LIN {X 0,Y 531.689,Z 306.036,A -85,B 0,C 180,E1 -12408.025,E2 -12408.025} C_VEL
LIN {X 0,Y 532.724,Z 312.75,A -85,B 0,C 180,E1 -12409.009,E2 -12409.009} C_VEL
LIN {X 0,Y 532.011,Z 332.528,A -85,B 0,C 180,E1 -12411.673,E2 -12411.673} C_VEL
LIN {X 0,Y 531.413,Z 343.977,A -85,B 0,C 180,E1 -12413.211,E2 -12413.211} C_VEL
LIN {X 0,Y 535.372,Z 363.328,A -85,B 0,C 180,E1 -12413.779,E2 -12413.779} C_VEL
LIN {X 0,Y 535.914,Z 368.587,A -85,B 0,C 180,E1 -12413.901,E2 -12413.901} C_VEL
LIN {X 0,Y 533.373,Z 483.364,A -85,B 0,C 180,E1 -12415.834,E2 -12415.834} C_VEL
LIN {X 0,Y 532.938,Z 496.517,A -85,B 0,C 180,E1 -12416.185,E2 -12416.185} C_VEL
LIN {X 0,Y 532.3,Z 510.41,A -85,B 0,C 180,E1 -12416.7,E2 -12416.7} C_VEL
LIN {X 0,Y 531.549,Z 523.766,A -85,B 0,C 180,E1 -12417.356,E2 -12417.356} C_VEL
LIN {X 0,Y 530.723,Z 537.278,A -85,B 0,C 180,E1 -12418.204,E2 -12418.204} C_VEL
LIN {X 0,Y 530.002,Z 549.395,A -85,B 0,C 180,E1 -12419.148,E2 -12419.148} C_VEL
LIN {X 0,Y 529.271,Z 560.359,A -85,B 0,C 180,E1 -12420.19,E2 -12420.19} C_VEL
LIN {X 0,Y 528.45,Z 570.244,A -85,B 0,C 180,E1 -12421.329,E2 -12421.329} C_VEL
LIN {X 0,Y 527.937,Z 578.439,A -85,B 0,C 180,E1 -12422.471,E2 -12422.471} C_VEL
LIN {X 0,Y 527.304,Z 586.33,A -85,B 0,C 180,E1 -12423.808,E2 -12423.808} C_VEL
LIN {X 0,Y 527.137,Z 592.304,A -85,B 0,C 180,E1 -12425.069,E2 -12425.069} C_VEL
LIN {X 0,Y 526.86,Z 597.604,A -85,B 0,C 180,E1 -12426.489,E2 -12426.489} C_VEL
LIN {X 0,Y 526.635,Z 600.902,A -85,B 0,C 180,E1 -12427.643,E2 -12427.643} C_VEL
LIN {X 0,Y 526.518,Z 603.931,A -85,B 0,C 180,E1 -12429.186,E2 -12429.186} C_VEL
LIN {X 0,Y 526.532,Z 605.072,A -85,B 0,C 180,E1 -12430.122,E2 -12430.122} C_VEL
LIN {X 0,Y 526.386,Z 605.783,A -85,B 0,C 180,E1 -12431.514,E2 -12431.514} C_VEL
LIN {X 0,Y 526.422,Z 605.211,A -85,B 0,C 180,E1 -12433.073,E2 -12433.073} C_VEL
LIN {X 0,Y 526.485,Z 604.366,A -85,B 0,C 180,E1 -12433.856,E2 -12433.856} C_VEL
LIN {X 0,Y 526.464,Z 601.496,A -85,B 0,C 180,E1 -12435.432,E2 -12435.432} C_VEL
LIN {X 0,Y 526.634,Z 597.945,A -85,B 0,C 180,E1 -12436.735,E2 -12436.735} C_VEL
LIN {X 0,Y 526.797,Z 592.499,A -85,B 0,C 180,E1 -12438.208,E2 -12438.208} C_VEL
LIN {X 0,Y 527.092,Z 585.795,A -85,B 0,C 180,E1 -12439.606,E2 -12439.606} C_VEL
LIN {X 0,Y 527.375,Z 578.63,A -85,B 0,C 180,E1 -12440.811,E2 -12440.811} C_VEL
LIN {X 0,Y 527.804,Z 569.924,A -85,B 0,C 180,E1 -12442.018,E2 -12442.018} C_VEL
LIN {X 0,Y 528.251,Z 561.2,A -85,B 0,C 180,E1 -12443.027,E2 -12443.027} C_VEL
LIN {X 0,Y 528.805,Z 549.803,A -85,B 0,C 180,E1 -12444.126,E2 -12444.126} C_VEL
LIN {X 0,Y 529.395,Z 538.058,A -85,B 0,C 180,E1 -12445.049,E2 -12445.049} C_VEL
LIN {X 0,Y 529.964,Z 525.375,A -85,B 0,C 180,E1 -12445.859,E2 -12445.859} C_VEL
LIN {X 0,Y 530.502,Z 511.263,A -85,B 0,C 180,E1 -12446.571,E2 -12446.571} C_VEL
LIN {X 0,Y 531.036,Z 496.754,A -85,B 0,C 180,E1 -12447.122,E2 -12447.122} C_VEL
LIN {X 0,Y 531.473,Z 482.696,A -85,B 0,C 180,E1 -12447.492,E2 -12447.492} C_VEL
LIN {X 0,Y 532,Z 441.042,A -85,B 0,C 180,E1 -12448.158,E2 -12448.158} C_VEL
LIN {X 0,Y 533.18,Z 365.683,A -85,B 0,C 180,E1 -12449.341,E2 -12449.341} C_VEL
LIN {X 0,Y 529.804,Z 342.816,A -85,B 0,C 180,E1 -12449.818,E2 -12449.818} C_VEL
LIN {X 0,Y 530.545,Z 321.092,A -85,B 0,C 180,E1 -12452.772,E2 -12452.772} C_VEL
LIN {X 0,Y 530.956,Z 306.195,A -85,B 0,C 180,E1 -12454.801,E2 -12454.801} C_VEL
LIN {X 0,Y 528.109,Z 291.26,A -85,B 0,C 180,E1 -12456.975,E2 -12456.975} C_VEL
LIN {X 0,Y 528.019,Z 291.272,A -85,B 0,C 180,E1 -12460.542,E2 -12460.542} C_VEL
LIN {X 0,Y 528.035,Z 291.266,A -85,B 0,C 180,E1 -12463.147,E2 -12463.147} C_VEL
LIN {X 0,Y 528.039,Z 291.267,A -85,B 0,C 180,E1 -12465.751,E2 -12465.751} C_VEL
LIN {X 0,Y 528.006,Z 291.272,A -85,B 0,C 180,E1 -12468.447,E2 -12468.447} C_VEL
LIN {X 0,Y 528.007,Z 291.272,A -85,B 0,C 180,E1 -12470.448,E2 -12470.448} C_VEL
LIN {X 0,Y 528.003,Z 291.271,A -85,B 0,C 180,E1 -12473.345,E2 -12473.345} C_VEL
LIN {X 0,Y 528.015,Z 291.272,A -85,B 0,C 180,E1 -12476.139,E2 -12476.139} C_VEL
LIN {X 0,Y 528.027,Z 291.268,A -85,B 0,C 180,E1 -12478.844,E2 -12478.844} C_VEL
LIN {X 0,Y 528.044,Z 291.267,A -85,B 0,C 180,E1 -12481.474,E2 -12481.474} C_VEL
LIN {X 0,Y 528.033,Z 291.271,A -85,B 0,C 180,E1 -12484.426,E2 -12484.426} C_VEL
LIN {X 0,Y 528.049,Z 291.266,A -85,B 0,C 180,E1 -12487.375,E2 -12487.375} C_VEL
LIN {X 0,Y 528.097,Z 291.262,A -85,B 0,C 180,E1 -12490.341,E2 -12490.341} C_VEL
LIN {X 0,Y 528.112,Z 291.256,A -85,B 0,C 180,E1 -12493.033,E2 -12493.033} C_VEL
LIN {X 0,Y 528.145,Z 291.256,A -85,B 0,C 180,E1 -12496.187,E2 -12496.187} C_VEL
LIN {X 0,Y 528.184,Z 291.248,A -85,B 0,C 180,E1 -12499.299,E2 -12499.299} C_VEL
LIN {X 0,Y 528.157,Z 291.254,A -85,B 0,C 180,E1 -12501.366,E2 -12501.366} C_VEL
LIN {X 0,Y 527.564,Z 291.698,A -85,B 0,C 180,E1 -12501.79,E2 -12501.79} C_VEL
LIN {X 0,Y 525.624,Z 293.294,A -85,B 0,C 180,E1 -12502.31,E2 -12502.31} C_VEL
LIN {X 0,Y 522.705,Z 296.934,A -85,B 0,C 180,E1 -12503.052,E2 -12503.052} C_VEL
LIN {X 0,Y 522.358,Z 298.956,A -85,B 0,C 180,E1 -12503.438,E2 -12503.438} C_VEL
LIN {X 0,Y 522.688,Z 302.419,A -85,B 0,C 180,E1 -12504.109,E2 -12504.109} C_VEL
LIN {X 0,Y 526.705,Z 322.513,A -85,B 0,C 180,E1 -12504.513,E2 -12504.513} C_VEL
LIN {X 0,Y 525.362,Z 438.155,A -85,B 0,C 180,E1 -12506.104,E2 -12506.104} C_VEL
LIN {X 0,Y 525.036,Z 452.552,A -85,B 0,C 180,E1 -12506.461,E2 -12506.461} C_VEL
LIN {X 0,Y 524.637,Z 465.786,A -85,B 0,C 180,E1 -12506.937,E2 -12506.937} C_VEL
LIN {X 0,Y 524.177,Z 477.882,A -85,B 0,C 180,E1 -12507.509,E2 -12507.509} C_VEL
LIN {X 0,Y 523.685,Z 490.578,A -85,B 0,C 180,E1 -12508.274,E2 -12508.274} C_VEL
LIN {X 0,Y 522.854,Z 502.219,A -85,B 0,C 180,E1 -12509.135,E2 -12509.135} C_VEL
LIN {X 0,Y 522.337,Z 513.758,A -85,B 0,C 180,E1 -12510.19,E2 -12510.19} C_VEL
LIN {X 0,Y 521.576,Z 524.151,A -85,B 0,C 180,E1 -12511.345,E2 -12511.345} C_VEL
LIN {X 0,Y 521.072,Z 532.709,A -85,B 0,C 180,E1 -12512.502,E2 -12512.502} C_VEL
LIN {X 0,Y 520.501,Z 540.947,A -85,B 0,C 180,E1 -12513.856,E2 -12513.856} C_VEL
LIN {X 0,Y 520.355,Z 546.848,A -85,B 0,C 180,E1 -12515.058,E2 -12515.058} C_VEL
LIN {X 0,Y 520.006,Z 552.804,A -85,B 0,C 180,E1 -12516.572,E2 -12516.572} C_VEL
LIN {X 0,Y 519.812,Z 556.307,A -85,B 0,C 180,E1 -12517.742,E2 -12517.742} C_VEL
LIN {X 0,Y 519.665,Z 559.732,A -85,B 0,C 180,E1 -12519.306,E2 -12519.306} C_VEL
LIN {X 0,Y 519.617,Z 561.765,A -85,B 0,C 180,E1 -12520.876,E2 -12520.876} C_VEL
LIN {X 0,Y 519.579,Z 562.436,A -85,B 0,C 180,E1 -12522.454,E2 -12522.454} C_VEL
LIN {X 0,Y 519.752,Z 561.732,A -85,B 0,C 180,E1 -12524.037,E2 -12524.037} C_VEL
LIN {X 0,Y 519.824,Z 559.65,A -85,B 0,C 180,E1 -12525.632,E2 -12525.632} C_VEL
LIN {X 0,Y 520.132,Z 556.106,A -85,B 0,C 180,E1 -12527.231,E2 -12527.231} C_VEL
LIN {X 0,Y 520.572,Z 550.981,A -85,B 0,C 180,E1 -12528.838,E2 -12528.838} C_VEL
LIN {X 0,Y 520.988,Z 545.954,A -85,B 0,C 180,E1 -12530.047,E2 -12530.047} C_VEL
LIN {X 0,Y 521.631,Z 538.658,A -85,B 0,C 180,E1 -12531.461,E2 -12531.461} C_VEL
LIN {X 0,Y 522.329,Z 530.905,A -85,B 0,C 180,E1 -12532.68,E2 -12532.68} C_VEL
LIN {X 0,Y 523.135,Z 521.574,A -85,B 0,C 180,E1 -12533.89,E2 -12533.89} C_VEL
LIN {X 0,Y 523.977,Z 511.439,A -85,B 0,C 180,E1 -12534.975,E2 -12534.975} C_VEL
LIN {X 0,Y 524.812,Z 500.782,A -85,B 0,C 180,E1 -12535.917,E2 -12535.917} C_VEL
LIN {X 0,Y 525.608,Z 489.128,A -85,B 0,C 180,E1 -12536.764,E2 -12536.764} C_VEL
LIN {X 0,Y 526.392,Z 475.732,A -85,B 0,C 180,E1 -12537.54,E2 -12537.54} C_VEL
LIN {X 0,Y 526.995,Z 461.981,A -85,B 0,C 180,E1 -12538.151,E2 -12538.151} C_VEL
LIN {X 0,Y 527.442,Z 447.824,A -85,B 0,C 180,E1 -12538.609,E2 -12538.609} C_VEL
LIN {X 0,Y 527.775,Z 433.139,A -85,B 0,C 180,E1 -12538.914,E2 -12538.914} C_VEL
LIN {X 0,Y 529.257,Z 323.678,A -85,B 0,C 180,E1 -12540.425,E2 -12540.425} C_VEL
LIN {X 0,Y 525.582,Z 309.533,A -85,B 0,C 180,E1 -12540.791,E2 -12540.791} C_VEL
LIN {X 0,Y 523.148,Z 303.089,A -85,B 0,C 180,E1 -12541.011,E2 -12541.011} C_VEL
LIN {X 0,Y 520.962,Z 292.15,A -85,B 0,C 180,E1 -12543.364,E2 -12543.364} C_VEL
LIN {X 0,Y 520.966,Z 292.152,A -85,B 0,C 180,E1 -12546.267,E2 -12546.267} C_VEL
LIN {X 0,Y 520.926,Z 292.149,A -85,B 0,C 180,E1 -12548.751,E2 -12548.751} C_VEL
LIN {X 0,Y 520.959,Z 292.145,A -85,B 0,C 180,E1 -12551.207,E2 -12551.207} C_VEL
LIN {X 0,Y 520.971,Z 292.139,A -85,B 0,C 180,E1 -12554.354,E2 -12554.354} C_VEL
LIN {X 0,Y 520.97,Z 292.147,A -85,B 0,C 180,E1 -12556.71,E2 -12556.71} C_VEL
LIN {X 0,Y 520.955,Z 292.152,A -85,B 0,C 180,E1 -12559.806,E2 -12559.806} C_VEL
LIN {X 0,Y 520.989,Z 292.139,A -85,B 0,C 180,E1 -12562.771,E2 -12562.771} C_VEL
LIN {X 0,Y 520.958,Z 292.132,A -85,B 0,C 180,E1 -12565.097,E2 -12565.097} C_VEL
LIN {X 0,Y 520.98,Z 292.147,A -85,B 0,C 180,E1 -12567.884,E2 -12567.884} C_VEL
LIN {X 0,Y 520.997,Z 292.143,A -85,B 0,C 180,E1 -12571.053,E2 -12571.053} C_VEL
LIN {X 0,Y 520.984,Z 292.145,A -85,B 0,C 180,E1 -12573.662,E2 -12573.662} C_VEL
LIN {X 0,Y 520.989,Z 292.137,A -85,B 0,C 180,E1 -12576.213,E2 -12576.213} C_VEL
LIN {X 0,Y 520.998,Z 292.141,A -85,B 0,C 180,E1 -12578.716,E2 -12578.716} C_VEL
LIN {X 0,Y 520.984,Z 292.14,A -85,B 0,C 180,E1 -12581.175,E2 -12581.175} C_VEL
LIN {X 0,Y 521.006,Z 292.146,A -85,B 0,C 180,E1 -12583.601,E2 -12583.601} C_VEL
LIN {X 0,Y 521.078,Z 292.125,A -85,B 0,C 180,E1 -12585.998,E2 -12585.998} C_VEL
LIN {X 0,Y 521.11,Z 292.134,A -85,B 0,C 180,E1 -12589.153,E2 -12589.153} C_VEL
LIN {X 0,Y 521.141,Z 292.12,A -85,B 0,C 180,E1 -12592.276,E2 -12592.276} C_VEL
LIN {X 0,Y 521.169,Z 292.121,A -85,B 0,C 180,E1 -12594.602,E2 -12594.602} C_VEL
LIN {X 0,Y 521.202,Z 292.105,A -85,B 0,C 180,E1 -12596.147,E2 -12596.147} C_VEL
LIN {X 0,Y 521.307,Z 292.109,A -85,B 0,C 180,E1 -12599.23,E2 -12599.23} C_VEL
LIN {X 0,Y 521.162,Z 292.112,A -85,B 0,C 180,E1 -12601.54,E2 -12601.54} C_VEL
LIN {X 0,Y 521.233,Z 292.114,A -85,B 0,C 180,E1 -12604.625,E2 -12604.625} C_VEL
LIN {X 0,Y 521.159,Z 292.116,A -85,B 0,C 180,E1 -12606.948,E2 -12606.948} C_VEL
LIN {X 0,Y 521.132,Z 292.123,A -85,B 0,C 180,E1 -12610.063,E2 -12610.063} C_VEL
LIN {X 0,Y 521.077,Z 292.126,A -85,B 0,C 180,E1 -12612.42,E2 -12612.42} C_VEL
LIN {X 0,Y 521.083,Z 292.135,A -85,B 0,C 180,E1 -12614.797,E2 -12614.797} C_VEL
LIN {X 0,Y 521.032,Z 292.127,A -85,B 0,C 180,E1 -12618.011,E2 -12618.011} C_VEL
LIN {X 0,Y 521.011,Z 292.143,A -85,B 0,C 180,E1 -12620.459,E2 -12620.459} C_VEL
LIN {X 0,Y 520.973,Z 292.146,A -85,B 0,C 180,E1 -12622.949,E2 -12622.949} C_VEL
LIN {X 0,Y 520.97,Z 292.142,A -85,B 0,C 180,E1 -12625.741,E2 -12625.741} C_VEL
LIN {X 0,Y 520.963,Z 292.146,A -85,B 0,C 180,E1 -12628.072,E2 -12628.072} C_VEL
LIN {X 0,Y 521.021,Z 292.139,A -85,B 0,C 180,E1 -12630.721,E2 -12630.721} C_VEL
LIN {X 0,Y 521.003,Z 292.138,A -85,B 0,C 180,E1 -12633.541,E2 -12633.541} C_VEL
LIN {X 0,Y 521.045,Z 292.118,A -85,B 0,C 180,E1 -12636.263,E2 -12636.263} C_VEL
LIN {X 0,Y 520.995,Z 292.142,A -85,B 0,C 180,E1 -12639.189,E2 -12639.189} C_VEL
LIN {X 0,Y 521.001,Z 292.146,A -85,B 0,C 180,E1 -12642.238,E2 -12642.238} C_VEL
LIN {X 0,Y 520.984,Z 292.141,A -85,B 0,C 180,E1 -12645.444,E2 -12645.444} C_VEL
LIN {X 0,Y 521.023,Z 292.14,A -85,B 0,C 180,E1 -12647.768,E2 -12647.768} C_VEL
LIN {X 0,Y 520.997,Z 292.143,A -85,B 0,C 180,E1 -12650.814,E2 -12650.814} C_VEL
LIN {X 0,Y 521.052,Z 292.134,A -85,B 0,C 180,E1 -12653.763,E2 -12653.763} C_VEL
LIN {X 0,Y 521.001,Z 292.145,A -85,B 0,C 180,E1 -12656.553,E2 -12656.553} C_VEL
LIN {X 0,Y 520.991,Z 292.151,A -85,B 0,C 180,E1 -12659.367,E2 -12659.367} C_VEL
LIN {X 0,Y 521.033,Z 292.33,A -85,B 0,C 180,E1 -12660.987,E2 -12660.987} C_VEL
LIN {X 0,Y 523.961,Z 305.085,A -85,B 0,C 180,E1 -12663.149,E2 -12663.149} C_VEL
LIN {X 0,Y 525.996,Z 315.082,A -85,B 0,C 180,E1 -12664.78,E2 -12664.78} C_VEL
LIN {X 0,Y 524.695,Z 333.223,A -85,B 0,C 180,E1 -12667.433,E2 -12667.433} C_VEL
LIN {X 0,Y 523.121,Z 355.773,A -85,B 0,C 180,E1 -12670.669,E2 -12670.669} C_VEL
LIN {X 0,Y 522.95,Z 358.465,A -85,B 0,C 180,E1 -12671.046,E2 -12671.046} C_VEL
LIN {X 0,Y 527.376,Z 385.573,A -85,B 0,C 180,E1 -12671.625,E2 -12671.625} C_VEL
LIN {X 0,Y 528.446,Z 395.781,A -85,B 0,C 180,E1 -12671.815,E2 -12671.815} C_VEL
LIN {X 0,Y 527.126,Z 496.999,A -85,B 0,C 180,E1 -12673.229,E2 -12673.229} C_VEL
LIN {X 0,Y 526.491,Z 511.69,A -85,B 0,C 180,E1 -12673.59,E2 -12673.59} C_VEL
LIN {X 0,Y 525.684,Z 525.843,A -85,B 0,C 180,E1 -12674.101,E2 -12674.101} C_VEL
LIN {X 0,Y 524.835,Z 538.666,A -85,B 0,C 180,E1 -12674.719,E2 -12674.719} C_VEL
LIN {X 0,Y 523.931,Z 551.153,A -85,B 0,C 180,E1 -12675.485,E2 -12675.485} C_VEL
LIN {X 0,Y 522.95,Z 562.578,A -85,B 0,C 180,E1 -12676.347,E2 -12676.347} C_VEL
LIN {X 0,Y 521.999,Z 574.075,A -85,B 0,C 180,E1 -12677.408,E2 -12677.408} C_VEL
LIN {X 0,Y 521.301,Z 584.778,A -85,B 0,C 180,E1 -12678.62,E2 -12678.62} C_VEL
LIN {X 0,Y 520.514,Z 594.203,A -85,B 0,C 180,E1 -12679.927,E2 -12679.927} C_VEL
LIN {X 0,Y 520.021,Z 602.18,A -85,B 0,C 180,E1 -12681.286,E2 -12681.286} C_VEL
LIN {X 0,Y 519.692,Z 608.639,A -85,B 0,C 180,E1 -12682.646,E2 -12682.646} C_VEL
LIN {X 0,Y 519.534,Z 615.45,A -85,B 0,C 180,E1 -12684.199,E2 -12684.199} C_VEL
LIN {X 0,Y 519.498,Z 619.544,A -85,B 0,C 180,E1 -12685.362,E2 -12685.362} C_VEL
LIN {X 0,Y 519.438,Z 622.038,A -85,B 0,C 180,E1 -12686.256,E2 -12686.256} C_VEL
LIN {X 0,Y 519.484,Z 624.964,A -85,B 0,C 180,E1 -12687.684,E2 -12687.684} C_VEL
LIN {X 0,Y 519.489,Z 626.706,A -85,B 0,C 180,E1 -12689.229,E2 -12689.229} C_VEL
LIN {X 0,Y 519.482,Z 627.012,A -85,B 0,C 180,E1 -12690.774,E2 -12690.774} C_VEL
LIN {X 0,Y 519.483,Z 625.891,A -85,B 0,C 180,E1 -12692.32,E2 -12692.32} C_VEL
LIN {X 0,Y 519.472,Z 623.335,A -85,B 0,C 180,E1 -12693.868,E2 -12693.868} C_VEL
LIN {X 0,Y 519.559,Z 619.26,A -85,B 0,C 180,E1 -12695.417,E2 -12695.417} C_VEL
LIN {X 0,Y 519.737,Z 613.522,A -85,B 0,C 180,E1 -12696.968,E2 -12696.968} C_VEL
LIN {X 0,Y 519.985,Z 607.026,A -85,B 0,C 180,E1 -12698.328,E2 -12698.328} C_VEL
LIN {X 0,Y 520.522,Z 598.946,A -85,B 0,C 180,E1 -12699.685,E2 -12699.685} C_VEL
LIN {X 0,Y 521.067,Z 590.487,A -85,B 0,C 180,E1 -12700.849,E2 -12700.849} C_VEL
LIN {X 0,Y 521.705,Z 580.297,A -85,B 0,C 180,E1 -12702.013,E2 -12702.013} C_VEL
LIN {X 0,Y 522.421,Z 568.9,A -85,B 0,C 180,E1 -12703.078,E2 -12703.078} C_VEL
LIN {X 0,Y 523.282,Z 556.204,A -85,B 0,C 180,E1 -12704.043,E2 -12704.043} C_VEL
LIN {X 0,Y 524.105,Z 543.638,A -85,B 0,C 180,E1 -12704.811,E2 -12704.811} C_VEL
LIN {X 0,Y 524.871,Z 530.794,A -85,B 0,C 180,E1 -12705.432,E2 -12705.432} C_VEL
LIN {X 0,Y 525.386,Z 518.702,A -85,B 0,C 180,E1 -12705.888,E2 -12705.888} C_VEL
LIN {X 0,Y 525.959,Z 503.876,A -85,B 0,C 180,E1 -12706.288,E2 -12706.288} C_VEL
LIN {X 0,Y 528.444,Z 394.307,A -85,B 0,C 180,E1 -12708.18,E2 -12708.18} C_VEL
LIN {X 0,Y 525.994,Z 372.212,A -85,B 0,C 180,E1 -12708.723,E2 -12708.723} C_VEL
LIN {X 0,Y 523.096,Z 353.92,A -85,B 0,C 180,E1 -12709.252,E2 -12709.252} C_VEL
LIN {X 0,Y 522.506,Z 348.155,A -85,B 0,C 180,E1 -12709.526,E2 -12709.526} C_VEL
LIN {X 0,Y 523.84,Z 324.588,A -85,B 0,C 180,E1 -12712.817,E2 -12712.817} C_VEL
LIN {X 0,Y 524.643,Z 310.622,A -85,B 0,C 180,E1 -12714.789,E2 -12714.789} C_VEL
LIN {X 0,Y 521.084,Z 292.136,A -85,B 0,C 180,E1 -12717.651,E2 -12717.651} C_VEL
LIN {X 0,Y 520.993,Z 292.145,A -85,B 0,C 180,E1 -12720.725,E2 -12720.725} C_VEL
LIN {X 0,Y 520.961,Z 292.151,A -85,B 0,C 180,E1 -12723.529,E2 -12723.529} C_VEL
LIN {X 0,Y 520.979,Z 292.147,A -85,B 0,C 180,E1 -12726.27,E2 -12726.27} C_VEL
LIN {X 0,Y 520.942,Z 292.155,A -85,B 0,C 180,E1 -12729.196,E2 -12729.196} C_VEL
LIN {X 0,Y 520.962,Z 292.145,A -85,B 0,C 180,E1 -12732.243,E2 -12732.243} C_VEL
LIN {X 0,Y 520.991,Z 292.146,A -85,B 0,C 180,E1 -12735.445,E2 -12735.445} C_VEL
LIN {X 0,Y 520.977,Z 292.148,A -85,B 0,C 180,E1 -12738.845,E2 -12738.845} C_VEL
LIN {X 0,Y 520.962,Z 292.148,A -85,B 0,C 180,E1 -12741.795,E2 -12741.795} C_VEL
LIN {X 0,Y 520.992,Z 292.147,A -85,B 0,C 180,E1 -12744.682,E2 -12744.682} C_VEL
LIN {X 0,Y 520.954,Z 292.148,A -85,B 0,C 180,E1 -12747.465,E2 -12747.465} C_VEL
LIN {X 0,Y 521.02,Z 292.143,A -85,B 0,C 180,E1 -12750.171,E2 -12750.171} C_VEL
LIN {X 0,Y 521.024,Z 292.144,A -85,B 0,C 180,E1 -12752.801,E2 -12752.801} C_VEL
LIN {X 0,Y 521.03,Z 292.146,A -85,B 0,C 180,E1 -12756.088,E2 -12756.088} C_VEL
LIN {X 0,Y 521.03,Z 292.149,A -85,B 0,C 180,E1 -12758.717,E2 -12758.717} C_VEL
LIN {X 0,Y 521.015,Z 292.148,A -85,B 0,C 180,E1 -12761.177,E2 -12761.177} C_VEL
LIN {X 0,Y 521.019,Z 292.148,A -85,B 0,C 180,E1 -12763.601,E2 -12763.601} C_VEL
LIN {X 0,Y 521.123,Z 292.285,A -85,B 0,C 180,E1 -12765.414,E2 -12765.414} C_VEL
LIN {X 0,Y 524.335,Z 304.944,A -85,B 0,C 180,E1 -12767.404,E2 -12767.404} C_VEL
LIN {X 0,Y 525.963,Z 313.242,A -85,B 0,C 180,E1 -12768.672,E2 -12768.672} C_VEL
LIN {X 0,Y 525.421,Z 330.67,A -85,B 0,C 180,E1 -12771.047,E2 -12771.047} C_VEL
LIN {X 0,Y 524.762,Z 344.54,A -85,B 0,C 180,E1 -12772.896,E2 -12772.896} C_VEL
LIN {X 0,Y 528.951,Z 364.875,A -85,B 0,C 180,E1 -12773.499,E2 -12773.499} C_VEL
LIN {X 0,Y 529.406,Z 369.542,A -85,B 0,C 180,E1 -12773.609,E2 -12773.609} C_VEL
LIN {X 0,Y 526.683,Z 484.36,A -85,B 0,C 180,E1 -12775.59,E2 -12775.59} C_VEL
LIN {X 0,Y 526.238,Z 497.17,A -85,B 0,C 180,E1 -12775.945,E2 -12775.945} C_VEL
LIN {X 0,Y 525.552,Z 510.883,A -85,B 0,C 180,E1 -12776.466,E2 -12776.466} C_VEL
LIN {X 0,Y 524.796,Z 524.163,A -85,B 0,C 180,E1 -12777.131,E2 -12777.131} C_VEL
LIN {X 0,Y 523.934,Z 537.634,A -85,B 0,C 180,E1 -12777.989,E2 -12777.989} C_VEL
LIN {X 0,Y 523.16,Z 549.705,A -85,B 0,C 180,E1 -12778.945,E2 -12778.945} C_VEL
LIN {X 0,Y 522.377,Z 560.627,A -85,B 0,C 180,E1 -12780,E2 -12780} C_VEL
LIN {X 0,Y 521.503,Z 570.5,A -85,B 0,C 180,E1 -12781.154,E2 -12781.154} C_VEL
LIN {X 0,Y 520.879,Z 579.904,A -85,B 0,C 180,E1 -12782.505,E2 -12782.505} C_VEL
LIN {X 0,Y 520.246,Z 587.559,A -85,B 0,C 180,E1 -12783.86,E2 -12783.86} C_VEL
LIN {X 0,Y 520.094,Z 592.682,A -85,B 0,C 180,E1 -12784.983,E2 -12784.983} C_VEL
LIN {X 0,Y 519.821,Z 597.184,A -85,B 0,C 180,E1 -12786.188,E2 -12786.188} C_VEL
LIN {X 0,Y 519.53,Z 601.545,A -85,B 0,C 180,E1 -12787.748,E2 -12787.748} C_VEL
LIN {X 0,Y 519.428,Z 604.395,A -85,B 0,C 180,E1 -12789.312,E2 -12789.312} C_VEL
LIN {X 0,Y 519.439,Z 605.317,A -85,B 0,C 180,E1 -12790.136,E2 -12790.136} C_VEL
LIN {X 0,Y 519.289,Z 605.965,A -85,B 0,C 180,E1 -12791.673,E2 -12791.673} C_VEL
LIN {X 0,Y 519.342,Z 605.151,A -85,B 0,C 180,E1 -12793.255,E2 -12793.255} C_VEL
LIN {X 0,Y 519.363,Z 604.189,A -85,B 0,C 180,E1 -12794.049,E2 -12794.049} C_VEL
LIN {X 0,Y 519.402,Z 601.119,A -85,B 0,C 180,E1 -12795.647,E2 -12795.647} C_VEL
LIN {X 0,Y 519.538,Z 597.864,A -85,B 0,C 180,E1 -12796.815,E2 -12796.815} C_VEL
LIN {X 0,Y 519.674,Z 593.388,A -85,B 0,C 180,E1 -12798.06,E2 -12798.06} C_VEL
LIN {X 0,Y 519.966,Z 587.04,A -85,B 0,C 180,E1 -12799.441,E2 -12799.441} C_VEL
LIN {X 0,Y 520.231,Z 579.882,A -85,B 0,C 180,E1 -12800.697,E2 -12800.697} C_VEL
LIN {X 0,Y 520.671,Z 571.447,A -85,B 0,C 180,E1 -12801.913,E2 -12801.913} C_VEL
LIN {X 0,Y 521.227,Z 561.052,A -85,B 0,C 180,E1 -12803.146,E2 -12803.146} C_VEL
LIN {X 0,Y 521.749,Z 550.448,A -85,B 0,C 180,E1 -12804.182,E2 -12804.182} C_VEL
LIN {X 0,Y 522.333,Z 539.177,A -85,B 0,C 180,E1 -12805.093,E2 -12805.093} C_VEL
LIN {X 0,Y 522.89,Z 526.716,A -85,B 0,C 180,E1 -12805.915,E2 -12805.915} C_VEL
LIN {X 0,Y 523.467,Z 513.002,A -85,B 0,C 180,E1 -12806.632,E2 -12806.632} C_VEL
LIN {X 0,Y 523.984,Z 498.898,A -85,B 0,C 180,E1 -12807.194,E2 -12807.194} C_VEL
LIN {X 0,Y 524.476,Z 484.73,A -85,B 0,C 180,E1 -12807.597,E2 -12807.597} C_VEL
LIN {X 0,Y 524.789,Z 465.494,A -85,B 0,C 180,E1 -12807.936,E2 -12807.936} C_VEL
LIN {X 0,Y 526.29,Z 366.439,A -85,B 0,C 180,E1 -12809.511,E2 -12809.511} C_VEL
LIN {X 0,Y 522.864,Z 342.96,A -85,B 0,C 180,E1 -12810.002,E2 -12810.002} C_VEL
LIN {X 0,Y 523.707,Z 319.224,A -85,B 0,C 180,E1 -12813.255,E2 -12813.255} C_VEL
LIN {X 0,Y 524.032,Z 307.627,A -85,B 0,C 180,E1 -12814.849,E2 -12814.849} C_VEL
LIN {X 0,Y 521.048,Z 292.14,A -85,B 0,C 180,E1 -12817.115,E2 -12817.115} C_VEL
LIN {X 0,Y 520.971,Z 292.151,A -85,B 0,C 180,E1 -12820.193,E2 -12820.193} C_VEL
LIN {X 0,Y 520.994,Z 292.142,A -85,B 0,C 180,E1 -12823.288,E2 -12823.288} C_VEL
LIN {X 0,Y 520.992,Z 292.144,A -85,B 0,C 180,E1 -12825.643,E2 -12825.643} C_VEL
LIN {X 0,Y 520.977,Z 292.147,A -85,B 0,C 180,E1 -12828.843,E2 -12828.843} C_VEL
LIN {X 0,Y 520.934,Z 292.153,A -85,B 0,C 180,E1 -12831.791,E2 -12831.791} C_VEL
LIN {X 0,Y 520.967,Z 292.149,A -85,B 0,C 180,E1 -12834.679,E2 -12834.679} C_VEL
LIN {X 0,Y 520.952,Z 292.149,A -85,B 0,C 180,E1 -12837.463,E2 -12837.463} C_VEL
LIN {X 0,Y 521.016,Z 292.144,A -85,B 0,C 180,E1 -12840.169,E2 -12840.169} C_VEL
LIN {X 0,Y 521.009,Z 292.142,A -85,B 0,C 180,E1 -12842.798,E2 -12842.798} C_VEL
LIN {X 0,Y 521.028,Z 292.143,A -85,B 0,C 180,E1 -12846.087,E2 -12846.087} C_VEL
LIN {X 0,Y 521.027,Z 292.14,A -85,B 0,C 180,E1 -12848.715,E2 -12848.715} C_VEL
LIN {X 0,Y 521.018,Z 292.14,A -85,B 0,C 180,E1 -12851.175,E2 -12851.175} C_VEL
LIN {X 0,Y 521.055,Z 292.137,A -85,B 0,C 180,E1 -12853.601,E2 -12853.601} C_VEL
LIN {X 0,Y 521.101,Z 292.136,A -85,B 0,C 180,E1 -12855.997,E2 -12855.997} C_VEL
LIN {X 0,Y 521.139,Z 292.124,A -85,B 0,C 180,E1 -12859.152,E2 -12859.152} C_VEL
LIN {X 0,Y 521.158,Z 292.127,A -85,B 0,C 180,E1 -12862.08,E2 -12862.08} C_VEL
LIN {X 0,Y 522.358,Z 298.956,A -85,B 0,C 180,E1 -12863.438,E2 -12863.438} C_VEL
LIN {X 0,Y 522.505,Z 301.37,A -85,B 0,C 180,E1 -12863.744,E2 -12863.744} C_VEL
LIN {X 0,Y 522.349,Z 305.552,A -85,B 0,C 180,E1 -12864.006,E2 -12864.006} C_VEL
LIN {X 0,Y 521.97,Z 309.844,A -85,B 0,C 180,E1 -12864.15,E2 -12864.15} C_VEL
LIN {X 0,Y 521.189,Z 316.099,A -85,B 0,C 180,E1 -12864.26,E2 -12864.26} C_VEL
LIN {X 0,Y 519.916,Z 325.393,A -85,B 0,C 180,E1 -12864.351,E2 -12864.351} C_VEL
LIN {X 0,Y 519.808,Z 329.127,A -85,B 0,C 180,E1 -12864.402,E2 -12864.402} C_VEL
LIN {X 0,Y 518.457,Z 438.742,A -85,B 0,C 180,E1 -12865.931,E2 -12865.931} C_VEL
LIN {X 0,Y 518.136,Z 453.07,A -85,B 0,C 180,E1 -12866.292,E2 -12866.292} C_VEL
LIN {X 0,Y 517.669,Z 466.849,A -85,B 0,C 180,E1 -12866.799,E2 -12866.799} C_VEL
LIN {X 0,Y 517.157,Z 480.53,A -85,B 0,C 180,E1 -12867.475,E2 -12867.475} C_VEL
LIN {X 0,Y 516.575,Z 492.821,A -85,B 0,C 180,E1 -12868.25,E2 -12868.25} C_VEL
LIN {X 0,Y 515.731,Z 505.283,A -85,B 0,C 180,E1 -12869.22,E2 -12869.22} C_VEL
LIN {X 0,Y 515.27,Z 515.411,A -85,B 0,C 180,E1 -12870.193,E2 -12870.193} C_VEL
LIN {X 0,Y 514.493,Z 525.573,A -85,B 0,C 180,E1 -12871.363,E2 -12871.363} C_VEL
LIN {X 0,Y 514.015,Z 533.961,A -85,B 0,C 180,E1 -12872.536,E2 -12872.536} C_VEL
LIN {X 0,Y 513.468,Z 540.975,A -85,B 0,C 180,E1 -12873.713,E2 -12873.713} C_VEL
LIN {X 0,Y 513.298,Z 547.372,A -85,B 0,C 180,E1 -12875.026,E2 -12875.026} C_VEL
LIN {X 0,Y 512.985,Z 552.268,A -85,B 0,C 180,E1 -12876.269,E2 -12876.269} C_VEL
LIN {X 0,Y 512.703,Z 557.066,A -85,B 0,C 180,E1 -12877.85,E2 -12877.85} C_VEL
LIN {X 0,Y 512.573,Z 560.374,A -85,B 0,C 180,E1 -12879.436,E2 -12879.436} C_VEL
LIN {X 0,Y 512.523,Z 562.275,A -85,B 0,C 180,E1 -12881.028,E2 -12881.028} C_VEL
LIN {X 0,Y 512.507,Z 562.828,A -85,B 0,C 180,E1 -12882.629,E2 -12882.629} C_VEL
LIN {X 0,Y 512.691,Z 562.019,A -85,B 0,C 180,E1 -12884.234,E2 -12884.234} C_VEL
LIN {X 0,Y 512.777,Z 559.831,A -85,B 0,C 180,E1 -12885.852,E2 -12885.852} C_VEL
LIN {X 0,Y 513.122,Z 556.175,A -85,B 0,C 180,E1 -12887.474,E2 -12887.474} C_VEL
LIN {X 0,Y 513.617,Z 550.93,A -85,B 0,C 180,E1 -12889.103,E2 -12889.103} C_VEL
LIN {X 0,Y 514.054,Z 545.772,A -85,B 0,C 180,E1 -12890.33,E2 -12890.33} C_VEL
LIN {X 0,Y 514.761,Z 538.336,A -85,B 0,C 180,E1 -12891.762,E2 -12891.762} C_VEL
LIN {X 0,Y 515.491,Z 530.454,A -85,B 0,C 180,E1 -12892.993,E2 -12892.993} C_VEL
LIN {X 0,Y 516.344,Z 521.033,A -85,B 0,C 180,E1 -12894.207,E2 -12894.207} C_VEL
LIN {X 0,Y 517.296,Z 510.152,A -85,B 0,C 180,E1 -12895.352,E2 -12895.352} C_VEL
LIN {X 0,Y 518.152,Z 499.525,A -85,B 0,C 180,E1 -12896.275,E2 -12896.275} C_VEL
LIN {X 0,Y 518.934,Z 488.184,A -85,B 0,C 180,E1 -12897.088,E2 -12897.088} C_VEL
LIN {X 0,Y 519.71,Z 475.543,A -85,B 0,C 180,E1 -12897.815,E2 -12897.815} C_VEL
LIN {X 0,Y 520.337,Z 461.614,A -85,B 0,C 180,E1 -12898.435,E2 -12898.435} C_VEL
LIN {X 0,Y 520.788,Z 448.031,A -85,B 0,C 180,E1 -12898.874,E2 -12898.874} C_VEL
LIN {X 0,Y 521.096,Z 434.638,A -85,B 0,C 180,E1 -12899.16,E2 -12899.16} C_VEL
LIN {X 0,Y 522.684,Z 325.067,A -85,B 0,C 180,E1 -12900.694,E2 -12900.694} C_VEL
LIN {X 0,Y 519.363,Z 312.13,A -85,B 0,C 180,E1 -12901.034,E2 -12901.034} C_VEL
LIN {X 0,Y 516.059,Z 303.611,A -85,B 0,C 180,E1 -12901.314,E2 -12901.314} C_VEL
LIN {X 0,Y 513.91,Z 293.03,A -85,B 0,C 180,E1 -12903.617,E2 -12903.617} C_VEL
LIN {X 0,Y 513.923,Z 293.026,A -85,B 0,C 180,E1 -12906.845,E2 -12906.845} C_VEL
LIN {X 0,Y 513.904,Z 293.03,A -85,B 0,C 180,E1 -12909.834,E2 -12909.834} C_VEL
LIN {X 0,Y 513.93,Z 293.025,A -85,B 0,C 180,E1 -12912.954,E2 -12912.954} C_VEL
LIN {X 0,Y 513.934,Z 293.026,A -85,B 0,C 180,E1 -12916.244,E2 -12916.244} C_VEL
LIN {X 0,Y 513.911,Z 293.026,A -85,B 0,C 180,E1 -12919.139,E2 -12919.139} C_VEL
LIN {X 0,Y 513.948,Z 293.02,A -85,B 0,C 180,E1 -12922.225,E2 -12922.225} C_VEL
LIN {X 0,Y 513.917,Z 293.008,A -85,B 0,C 180,E1 -12924.858,E2 -12924.858} C_VEL
LIN {X 0,Y 513.95,Z 293.023,A -85,B 0,C 180,E1 -12927.892,E2 -12927.892} C_VEL
LIN {X 0,Y 513.954,Z 293.019,A -85,B 0,C 180,E1 -12930.713,E2 -12930.713} C_VEL
LIN {X 0,Y 513.957,Z 293.015,A -85,B 0,C 180,E1 -12933.273,E2 -12933.273} C_VEL
LIN {X 0,Y 513.946,Z 293.017,A -85,B 0,C 180,E1 -12935.934,E2 -12935.934} C_VEL
LIN {X 0,Y 513.963,Z 293.018,A -85,B 0,C 180,E1 -12938.41,E2 -12938.41} C_VEL
LIN {X 0,Y 513.941,Z 293.017,A -85,B 0,C 180,E1 -12940.908,E2 -12940.908} C_VEL
LIN {X 0,Y 513.951,Z 293.025,A -85,B 0,C 180,E1 -12943.369,E2 -12943.369} C_VEL
LIN {X 0,Y 514.046,Z 293.002,A -85,B 0,C 180,E1 -12945.802,E2 -12945.802} C_VEL
LIN {X 0,Y 514.064,Z 293.009,A -85,B 0,C 180,E1 -12949.003,E2 -12949.003} C_VEL
LIN {X 0,Y 514.09,Z 292.998,A -85,B 0,C 180,E1 -12952.169,E2 -12952.169} C_VEL
LIN {X 0,Y 514.194,Z 292.986,A -85,B 0,C 180,E1 -12955.312,E2 -12955.312} C_VEL
LIN {X 0,Y 514.255,Z 292.987,A -85,B 0,C 180,E1 -12959.22,E2 -12959.22} C_VEL
LIN {X 0,Y 514.109,Z 292.99,A -85,B 0,C 180,E1 -12961.561,E2 -12961.561} C_VEL
LIN {X 0,Y 514.203,Z 292.991,A -85,B 0,C 180,E1 -12964.688,E2 -12964.688} C_VEL
LIN {X 0,Y 514.092,Z 292.993,A -85,B 0,C 180,E1 -12967.831,E2 -12967.831} C_VEL
LIN {X 0,Y 514.128,Z 292.993,A -85,B 0,C 180,E1 -12971.224,E2 -12971.224} C_VEL
LIN {X 0,Y 514.057,Z 293.007,A -85,B 0,C 180,E1 -12974.674,E2 -12974.674} C_VEL
LIN {X 0,Y 514.015,Z 293.002,A -85,B 0,C 180,E1 -12977.477,E2 -12977.477} C_VEL
LIN {X 0,Y 513.973,Z 293.018,A -85,B 0,C 180,E1 -12980.752,E2 -12980.752} C_VEL
LIN {X 0,Y 513.921,Z 293.023,A -85,B 0,C 180,E1 -12983.282,E2 -12983.282} C_VEL
LIN {X 0,Y 513.924,Z 293.02,A -85,B 0,C 180,E1 -12985.909,E2 -12985.909} C_VEL
LIN {X 0,Y 513.92,Z 293.029,A -85,B 0,C 180,E1 -12988.492,E2 -12988.492} C_VEL
LIN {X 0,Y 513.959,Z 293.018,A -85,B 0,C 180,E1 -12991.19,E2 -12991.19} C_VEL
LIN {X 0,Y 513.938,Z 293.02,A -85,B 0,C 180,E1 -12993.972,E2 -12993.972} C_VEL
LIN {X 0,Y 513.999,Z 293.004,A -85,B 0,C 180,E1 -12996.842,E2 -12996.842} C_VEL
LIN {X 0,Y 513.978,Z 293.018,A -85,B 0,C 180,E1 -13000.26,E2 -13000.26} C_VEL
LIN {X 0,Y 513.936,Z 293.021,A -85,B 0,C 180,E1 -13002.957,E2 -13002.957} C_VEL
LIN {X 0,Y 513.946,Z 293.023,A -85,B 0,C 180,E1 -13005.971,E2 -13005.971} C_VEL
LIN {X 0,Y 513.961,Z 293.021,A -85,B 0,C 180,E1 -13008.552,E2 -13008.552} C_VEL
LIN {X 0,Y 513.946,Z 293.02,A -85,B 0,C 180,E1 -13011.18,E2 -13011.18} C_VEL
LIN {X 0,Y 513.971,Z 293.019,A -85,B 0,C 180,E1 -13014.129,E2 -13014.129} C_VEL
LIN {X 0,Y 513.96,Z 293.025,A -85,B 0,C 180,E1 -13016.969,E2 -13016.969} C_VEL
LIN {X 0,Y 513.944,Z 293.031,A -85,B 0,C 180,E1 -13019.72,E2 -13019.72} C_VEL
LIN {X 0,Y 513.976,Z 293.04,A -85,B 0,C 180,E1 -13020.665,E2 -13020.665} C_VEL
LIN {X 0,Y 517.086,Z 306.623,A -85,B 0,C 180,E1 -13023.009,E2 -13023.009} C_VEL
LIN {X 0,Y 519.141,Z 316.735,A -85,B 0,C 180,E1 -13024.688,E2 -13024.688} C_VEL
LIN {X 0,Y 517.792,Z 334.559,A -85,B 0,C 180,E1 -13027.326,E2 -13027.326} C_VEL
LIN {X 0,Y 516.266,Z 355.648,A -85,B 0,C 180,E1 -13030.402,E2 -13030.402} C_VEL
LIN {X 0,Y 516.102,Z 358.24,A -85,B 0,C 180,E1 -13030.741,E2 -13030.741} C_VEL
LIN {X 0,Y 520.712,Z 386.02,A -85,B 0,C 180,E1 -13031.351,E2 -13031.351} C_VEL
LIN {X 0,Y 521.815,Z 396.677,A -85,B 0,C 180,E1 -13031.553,E2 -13031.553} C_VEL
LIN {X 0,Y 520.433,Z 496.846,A -85,B 0,C 180,E1 -13032.972,E2 -13032.972} C_VEL
LIN {X 0,Y 519.796,Z 511.094,A -85,B 0,C 180,E1 -13033.325,E2 -13033.325} C_VEL
LIN {X 0,Y 519.051,Z 524.087,A -85,B 0,C 180,E1 -13033.791,E2 -13033.791} C_VEL
LIN {X 0,Y 518.114,Z 537.201,A -85,B 0,C 180,E1 -13034.416,E2 -13034.416} C_VEL
LIN {X 0,Y 517.139,Z 549.889,A -85,B 0,C 180,E1 -13035.19,E2 -13035.19} C_VEL
LIN {X 0,Y 516.143,Z 561.462,A -85,B 0,C 180,E1 -13036.064,E2 -13036.064} C_VEL
LIN {X 0,Y 515.234,Z 572.101,A -85,B 0,C 180,E1 -13037.04,E2 -13037.04} C_VEL
LIN {X 0,Y 514.442,Z 582.681,A -85,B 0,C 180,E1 -13038.217,E2 -13038.217} C_VEL
LIN {X 0,Y 513.771,Z 591.446,A -85,B 0,C 180,E1 -13039.396,E2 -13039.396} C_VEL
LIN {X 0,Y 513.124,Z 599.885,A -85,B 0,C 180,E1 -13040.772,E2 -13040.772} C_VEL
LIN {X 0,Y 512.677,Z 606.707,A -85,B 0,C 180,E1 -13042.149,E2 -13042.149} C_VEL
LIN {X 0,Y 512.452,Z 616.553,A -85,B 0,C 180,E1 -13044.512,E2 -13044.512} C_VEL
LIN {X 0,Y 512.38,Z 621.457,A -85,B 0,C 180,E1 -13046.083,E2 -13046.083} C_VEL
LIN {X 0,Y 512.401,Z 624.734,A -85,B 0,C 180,E1 -13047.652,E2 -13047.652} C_VEL
LIN {X 0,Y 512.416,Z 626.522,A -85,B 0,C 180,E1 -13049.219,E2 -13049.219} C_VEL
LIN {X 0,Y 512.409,Z 626.872,A -85,B 0,C 180,E1 -13050.785,E2 -13050.785} C_VEL
LIN {X 0,Y 512.381,Z 625.792,A -85,B 0,C 180,E1 -13052.352,E2 -13052.352} C_VEL
LIN {X 0,Y 512.383,Z 623.273,A -85,B 0,C 180,E1 -13053.921,E2 -13053.921} C_VEL
LIN {X 0,Y 512.475,Z 619.252,A -85,B 0,C 180,E1 -13055.492,E2 -13055.492} C_VEL
LIN {X 0,Y 512.675,Z 613.564,A -85,B 0,C 180,E1 -13057.065,E2 -13057.065} C_VEL
LIN {X 0,Y 512.947,Z 607.124,A -85,B 0,C 180,E1 -13058.443,E2 -13058.443} C_VEL
LIN {X 0,Y 513.518,Z 599.082,A -85,B 0,C 180,E1 -13059.819,E2 -13059.819} C_VEL
LIN {X 0,Y 514.103,Z 590.677,A -85,B 0,C 180,E1 -13060.998,E2 -13060.998} C_VEL
LIN {X 0,Y 514.785,Z 580.573,A -85,B 0,C 180,E1 -13062.177,E2 -13062.177} C_VEL
LIN {X 0,Y 515.53,Z 569.331,A -85,B 0,C 180,E1 -13063.256,E2 -13063.256} C_VEL
LIN {X 0,Y 516.435,Z 556.747,A -85,B 0,C 180,E1 -13064.233,E2 -13064.233} C_VEL
LIN {X 0,Y 517.279,Z 544.349,A -85,B 0,C 180,E1 -13065.011,E2 -13065.011} C_VEL
LIN {X 0,Y 518.135,Z 530.697,A -85,B 0,C 180,E1 -13065.688,E2 -13065.688} C_VEL
LIN {X 0,Y 518.774,Z 517.972,A -85,B 0,C 180,E1 -13066.171,E2 -13066.171} C_VEL
LIN {X 0,Y 519.322,Z 503.712,A -85,B 0,C 180,E1 -13066.561,E2 -13066.561} C_VEL
LIN {X 0,Y 521.956,Z 395.263,A -85,B 0,C 180,E1 -13068.476,E2 -13068.476} C_VEL
LIN {X 0,Y 519.652,Z 373.978,A -85,B 0,C 180,E1 -13069.012,E2 -13069.012} C_VEL
LIN {X 0,Y 516.566,Z 353.92,A -85,B 0,C 180,E1 -13069.605,E2 -13069.605} C_VEL
LIN {X 0,Y 515.622,Z 346.225,A -85,B 0,C 180,E1 -13069.974,E2 -13069.974} C_VEL
LIN {X 0,Y 516.954,Z 323.892,A -85,B 0,C 180,E1 -13073.139,E2 -13073.139} C_VEL
LIN {X 0,Y 517.7,Z 312.263,A -85,B 0,C 180,E1 -13074.8,E2 -13074.8} C_VEL
LIN {X 0,Y 514.041,Z 293.011,A -85,B 0,C 180,E1 -13077.8,E2 -13077.8} C_VEL
LIN {X 0,Y 513.937,Z 293.023,A -85,B 0,C 180,E1 -13080.837,E2 -13080.837} C_VEL
LIN {X 0,Y 513.922,Z 293.028,A -85,B 0,C 180,E1 -13083.975,E2 -13083.975} C_VEL
LIN {X 0,Y 513.923,Z 293.026,A -85,B 0,C 180,E1 -13086.85,E2 -13086.85} C_VEL
LIN {X 0,Y 513.927,Z 293.024,A -85,B 0,C 180,E1 -13090.249,E2 -13090.249} C_VEL
LIN {X 0,Y 513.917,Z 293.026,A -85,B 0,C 180,E1 -13092.961,E2 -13092.961} C_VEL
LIN {X 0,Y 513.946,Z 293.021,A -85,B 0,C 180,E1 -13096.248,E2 -13096.248} C_VEL
LIN {X 0,Y 513.923,Z 293.029,A -85,B 0,C 180,E1 -13099.14,E2 -13099.14} C_VEL
LIN {X 0,Y 513.966,Z 293.021,A -85,B 0,C 180,E1 -13102.228,E2 -13102.228} C_VEL
LIN {X 0,Y 513.942,Z 293.025,A -85,B 0,C 180,E1 -13105.081,E2 -13105.081} C_VEL
LIN {X 0,Y 513.935,Z 293.023,A -85,B 0,C 180,E1 -13107.891,E2 -13107.891} C_VEL
LIN {X 0,Y 513.98,Z 293.022,A -85,B 0,C 180,E1 -13110.715,E2 -13110.715} C_VEL
LIN {X 0,Y 513.986,Z 293.018,A -85,B 0,C 180,E1 -13113.275,E2 -13113.275} C_VEL
LIN {X 0,Y 513.976,Z 293.025,A -85,B 0,C 180,E1 -13115.936,E2 -13115.936} C_VEL
LIN {X 0,Y 513.994,Z 293.027,A -85,B 0,C 180,E1 -13118.411,E2 -13118.411} C_VEL
LIN {X 0,Y 513.972,Z 293.027,A -85,B 0,C 180,E1 -13120.909,E2 -13120.909} C_VEL
LIN {X 0,Y 513.965,Z 293.025,A -85,B 0,C 180,E1 -13123.37,E2 -13123.37} C_VEL
LIN {X 0,Y 514.062,Z 293.154,A -85,B 0,C 180,E1 -13125.022,E2 -13125.022} C_VEL
LIN {X 0,Y 517.396,Z 306.05,A -85,B 0,C 180,E1 -13127.095,E2 -13127.095} C_VEL
LIN {X 0,Y 519.289,Z 315.292,A -85,B 0,C 180,E1 -13128.524,E2 -13128.524} C_VEL
LIN {X 0,Y 518.793,Z 330.876,A -85,B 0,C 180,E1 -13130.676,E2 -13130.676} C_VEL
LIN {X 0,Y 518.042,Z 344.551,A -85,B 0,C 180,E1 -13132.535,E2 -13132.535} C_VEL
LIN {X 0,Y 522.328,Z 365.047,A -85,B 0,C 180,E1 -13133.17,E2 -13133.17} C_VEL
LIN {X 0,Y 522.935,Z 369.874,A -85,B 0,C 180,E1 -13133.296,E2 -13133.296} C_VEL
LIN {X 0,Y 520.048,Z 484.269,A -85,B 0,C 180,E1 -13135.313,E2 -13135.313} C_VEL
LIN {X 0,Y 519.549,Z 497.997,A -85,B 0,C 180,E1 -13135.699,E2 -13135.699} C_VEL
LIN {X 0,Y 518.761,Z 512.525,A -85,B 0,C 180,E1 -13136.274,E2 -13136.274} C_VEL
LIN {X 0,Y 517.949,Z 526.287,A -85,B 0,C 180,E1 -13136.996,E2 -13136.996} C_VEL
LIN {X 0,Y 517.031,Z 539.393,A -85,B 0,C 180,E1 -13137.865,E2 -13137.865} C_VEL
LIN {X 0,Y 516.226,Z 551.141,A -85,B 0,C 180,E1 -13138.834,E2 -13138.834} C_VEL
LIN {X 0,Y 515.343,Z 562.688,A -85,B 0,C 180,E1 -13140,E2 -13140} C_VEL
LIN {X 0,Y 514.448,Z 572.257,A -85,B 0,C 180,E1 -13141.17,E2 -13141.17} C_VEL
LIN {X 0,Y 513.892,Z 580.174,A -85,B 0,C 180,E1 -13142.343,E2 -13142.343} C_VEL
LIN {X 0,Y 513.294,Z 586.808,A -85,B 0,C 180,E1 -13143.521,E2 -13143.521} C_VEL
LIN {X 0,Y 513.086,Z 592.437,A -85,B 0,C 180,E1 -13144.738,E2 -13144.738} C_VEL
LIN {X 0,Y 512.742,Z 598.028,A -85,B 0,C 180,E1 -13146.274,E2 -13146.274} C_VEL
LIN {X 0,Y 512.426,Z 602.198,A -85,B 0,C 180,E1 -13147.856,E2 -13147.856} C_VEL
LIN {X 0,Y 512.347,Z 604.849,A -85,B 0,C 180,E1 -13149.442,E2 -13149.442} C_VEL
LIN {X 0,Y 512.333,Z 605.616,A -85,B 0,C 180,E1 -13150.238,E2 -13150.238} C_VEL
LIN {X 0,Y 512.196,Z 606.069,A -85,B 0,C 180,E1 -13151.837,E2 -13151.837} C_VEL
LIN {X 0,Y 512.274,Z 605.06,A -85,B 0,C 180,E1 -13153.441,E2 -13153.441} C_VEL
LIN {X 0,Y 512.251,Z 602.557,A -85,B 0,C 180,E1 -13155.058,E2 -13155.058} C_VEL
LIN {X 0,Y 512.389,Z 599.621,A -85,B 0,C 180,E1 -13156.274,E2 -13156.274} C_VEL
LIN {X 0,Y 512.512,Z 595.733,A -85,B 0,C 180,E1 -13157.498,E2 -13157.498} C_VEL
LIN {X 0,Y 512.707,Z 590.797,A -85,B 0,C 180,E1 -13158.726,E2 -13158.726} C_VEL
LIN {X 0,Y 512.984,Z 584.677,A -85,B 0,C 180,E1 -13159.96,E2 -13159.96} C_VEL
LIN {X 0,Y 513.339,Z 577.184,A -85,B 0,C 180,E1 -13161.198,E2 -13161.198} C_VEL
LIN {X 0,Y 513.786,Z 568.034,A -85,B 0,C 180,E1 -13162.44,E2 -13162.44} C_VEL
LIN {X 0,Y 514.341,Z 557.872,A -85,B 0,C 180,E1 -13163.58,E2 -13163.58} C_VEL
LIN {X 0,Y 514.932,Z 546.75,A -85,B 0,C 180,E1 -13164.612,E2 -13164.612} C_VEL
LIN {X 0,Y 515.555,Z 534.383,A -85,B 0,C 180,E1 -13165.554,E2 -13165.554} C_VEL
LIN {X 0,Y 516.159,Z 521.811,A -85,B 0,C 180,E1 -13166.327,E2 -13166.327} C_VEL
LIN {X 0,Y 516.676,Z 508.873,A -85,B 0,C 180,E1 -13166.956,E2 -13166.956} C_VEL
LIN {X 0,Y 517.204,Z 494.811,A -85,B 0,C 180,E1 -13167.471,E2 -13167.471} C_VEL
LIN {X 0,Y 517.601,Z 479.461,A -85,B 0,C 180,E1 -13167.859,E2 -13167.859} C_VEL
LIN {X 0,Y 519.355,Z 367.003,A -85,B 0,C 180,E1 -13169.691,E2 -13169.691} C_VEL
LIN {X 0,Y 515.881,Z 342.999,A -85,B 0,C 180,E1 -13170.213,E2 -13170.213} C_VEL
LIN {X 0,Y 516.727,Z 320.625,A -85,B 0,C 180,E1 -13173.298,E2 -13173.298} C_VEL
LIN {X 0,Y 517.079,Z 308.957,A -85,B 0,C 180,E1 -13174.913,E2 -13174.913} C_VEL
LIN {X 0,Y 514.019,Z 293.015,A -85,B 0,C 180,E1 -13177.268,E2 -13177.268} C_VEL
LIN {X 0,Y 513.927,Z 293.025,A -85,B 0,C 180,E1 -13180.859,E2 -13180.859} C_VEL
LIN {X 0,Y 513.959,Z 293.02,A -85,B 0,C 180,E1 -13183.753,E2 -13183.753} C_VEL
LIN {X 0,Y 513.924,Z 293.024,A -85,B 0,C 180,E1 -13187.04,E2 -13187.04} C_VEL
LIN {X 0,Y 513.924,Z 293.028,A -85,B 0,C 180,E1 -13190.163,E2 -13190.163} C_VEL
LIN {X 0,Y 513.924,Z 293.025,A -85,B 0,C 180,E1 -13193.526,E2 -13193.526} C_VEL
LIN {X 0,Y 513.936,Z 293.026,A -85,B 0,C 180,E1 -13196.24,E2 -13196.24} C_VEL
LIN {X 0,Y 513.937,Z 293.022,A -85,B 0,C 180,E1 -13199.163,E2 -13199.163} C_VEL
LIN {X 0,Y 513.94,Z 293.023,A -85,B 0,C 180,E1 -13201.508,E2 -13201.508} C_VEL
LIN {X 0,Y 513.944,Z 293.025,A -85,B 0,C 180,E1 -13204.142,E2 -13204.142} C_VEL
LIN {X 0,Y 513.948,Z 293.021,A -85,B 0,C 180,E1 -13206.718,E2 -13206.718} C_VEL
LIN {X 0,Y 514.001,Z 293.014,A -85,B 0,C 180,E1 -13209.247,E2 -13209.247} C_VEL
LIN {X 0,Y 514.007,Z 293.014,A -85,B 0,C 180,E1 -13212.553,E2 -13212.553} C_VEL
LIN {X 0,Y 514.072,Z 293.009,A -85,B 0,C 180,E1 -13215.801,E2 -13215.801} C_VEL
LIN {X 0,Y 514.093,Z 293.001,A -85,B 0,C 180,E1 -13219.002,E2 -13219.002} C_VEL
LIN {X 0,Y 514.138,Z 293.155,A -85,B 0,C 180,E1 -13221.971,E2 -13221.971} C_VEL
LIN {X 0,Y 515.665,Z 302.712,A -85,B 0,C 180,E1 -13223.882,E2 -13223.882} C_VEL
LIN {X 0,Y 519.838,Z 323.214,A -85,B 0,C 180,E1 -13224.319,E2 -13224.319} C_VEL
LIN {X 0,Y 519.808,Z 329.127,A -85,B 0,C 180,E1 -13224.402,E2 -13224.402} C_VEL
LIN {X 0,Y 519.1,Z 334.966,A -85,B 0,C 180,E1 -13224.463,E2 -13224.463} C_VEL
LIN {X 0,Y 513.2,Z 353.902,A -85,B 0,C 180,E1 -13224.557,E2 -13224.557} C_VEL
LIN {X 0,Y 512.49,Z 359.742,A -85,B 0,C 180,E1 -13224.619,E2 -13224.619} C_VEL
LIN {X 0,Y 511.555,Z 439.33,A -85,B 0,C 180,E1 -13225.753,E2 -13225.753} C_VEL
LIN {X 0,Y 511.23,Z 453.594,A -85,B 0,C 180,E1 -13226.119,E2 -13226.119} C_VEL
LIN {X 0,Y 510.796,Z 466.773,A -85,B 0,C 180,E1 -13226.608,E2 -13226.608} C_VEL
LIN {X 0,Y 510.273,Z 479.701,A -85,B 0,C 180,E1 -13227.244,E2 -13227.244} C_VEL
LIN {X 0,Y 509.72,Z 492.212,A -85,B 0,C 180,E1 -13228.029,E2 -13228.029} C_VEL
LIN {X 0,Y 508.859,Z 503.709,A -85,B 0,C 180,E1 -13228.914,E2 -13228.914} C_VEL
LIN {X 0,Y 508.311,Z 515.135,A -85,B 0,C 180,E1 -13229.998,E2 -13229.998} C_VEL
LIN {X 0,Y 507.51,Z 525.436,A -85,B 0,C 180,E1 -13231.184,E2 -13231.184} C_VEL
LIN {X 0,Y 507.01,Z 533.912,A -85,B 0,C 180,E1 -13232.373,E2 -13232.373} C_VEL
LIN {X 0,Y 506.382,Z 542.062,A -85,B 0,C 180,E1 -13233.765,E2 -13233.765} C_VEL
LIN {X 0,Y 506.231,Z 547.836,A -85,B 0,C 180,E1 -13234.979,E2 -13234.979} C_VEL
LIN {X 0,Y 505.888,Z 553.138,A -85,B 0,C 180,E1 -13236.357,E2 -13236.357} C_VEL
LIN {X 0,Y 505.688,Z 556.752,A -85,B 0,C 180,E1 -13237.559,E2 -13237.559} C_VEL
LIN {X 0,Y 505.527,Z 559.568,A -85,B 0,C 180,E1 -13238.765,E2 -13238.765} C_VEL
LIN {X 0,Y 505.496,Z 562.038,A -85,B 0,C 180,E1 -13240.376,E2 -13240.376} C_VEL
LIN {X 0,Y 505.413,Z 563.164,A -85,B 0,C 180,E1 -13241.996,E2 -13241.996} C_VEL
LIN {X 0,Y 505.528,Z 562.933,A -85,B 0,C 180,E1 -13243.622,E2 -13243.622} C_VEL
LIN {X 0,Y 505.65,Z 561.339,A -85,B 0,C 180,E1 -13245.257,E2 -13245.257} C_VEL
LIN {X 0,Y 505.922,Z 558.319,A -85,B 0,C 180,E1 -13246.9,E2 -13246.9} C_VEL
LIN {X 0,Y 506.367,Z 553.766,A -85,B 0,C 180,E1 -13248.549,E2 -13248.549} C_VEL
LIN {X 0,Y 506.906,Z 548.294,A -85,B 0,C 180,E1 -13250.011,E2 -13250.011} C_VEL
LIN {X 0,Y 507.53,Z 541.441,A -85,B 0,C 180,E1 -13251.45,E2 -13251.45} C_VEL
LIN {X 0,Y 508.278,Z 534.144,A -85,B 0,C 180,E1 -13252.695,E2 -13252.695} C_VEL
LIN {X 0,Y 509.133,Z 525.272,A -85,B 0,C 180,E1 -13253.942,E2 -13253.942} C_VEL
LIN {X 0,Y 510.042,Z 515.466,A -85,B 0,C 180,E1 -13255.081,E2 -13255.081} C_VEL
LIN {X 0,Y 510.985,Z 504.569,A -85,B 0,C 180,E1 -13256.124,E2 -13256.124} C_VEL
LIN {X 0,Y 512.005,Z 491.792,A -85,B 0,C 180,E1 -13257.117,E2 -13257.117} C_VEL
LIN {X 0,Y 512.811,Z 479.358,A -85,B 0,C 180,E1 -13257.89,E2 -13257.89} C_VEL
LIN {X 0,Y 513.527,Z 465.371,A -85,B 0,C 180,E1 -13258.568,E2 -13258.568} C_VEL
LIN {X 0,Y 514.084,Z 451.312,A -85,B 0,C 180,E1 -13259.063,E2 -13259.063} C_VEL
LIN {X 0,Y 514.43,Z 438.349,A -85,B 0,C 180,E1 -13259.376,E2 -13259.376} C_VEL
LIN {X 0,Y 516.019,Z 325.71,A -85,B 0,C 180,E1 -13260.987,E2 -13260.987} C_VEL
LIN {X 0,Y 513.132,Z 314.686,A -85,B 0,C 180,E1 -13261.285,E2 -13261.285} C_VEL
LIN {X 0,Y 508.961,Z 303.93,A -85,B 0,C 180,E1 -13261.663,E2 -13261.663} C_VEL
LIN {X 0,Y 506.879,Z 293.908,A -85,B 0,C 180,E1 -13263.885,E2 -13263.885} C_VEL
LIN {X 0,Y 506.9,Z 293.902,A -85,B 0,C 180,E1 -13266.731,E2 -13266.731} C_VEL
LIN {X 0,Y 506.845,Z 293.905,A -85,B 0,C 180,E1 -13269.469,E2 -13269.469} C_VEL
LIN {X 0,Y 506.907,Z 293.9,A -85,B 0,C 180,E1 -13272.916,E2 -13272.916} C_VEL
LIN {X 0,Y 506.91,Z 293.902,A -85,B 0,C 180,E1 -13276.299,E2 -13276.299} C_VEL
LIN {X 0,Y 506.863,Z 293.907,A -85,B 0,C 180,E1 -13279.496,E2 -13279.496} C_VEL
LIN {X 0,Y 506.905,Z 293.894,A -85,B 0,C 180,E1 -13282.555,E2 -13282.555} C_VEL
LIN {X 0,Y 506.874,Z 293.889,A -85,B 0,C 180,E1 -13285.488,E2 -13285.488} C_VEL
LIN {X 0,Y 506.898,Z 293.896,A -85,B 0,C 180,E1 -13288.325,E2 -13288.325} C_VEL
LIN {X 0,Y 506.881,Z 293.902,A -85,B 0,C 180,E1 -13291.076,E2 -13291.076} C_VEL
LIN {X 0,Y 506.878,Z 293.905,A -85,B 0,C 180,E1 -13293.919,E2 -13293.919} C_VEL
LIN {X 0,Y 506.875,Z 293.894,A -85,B 0,C 180,E1 -13296.375,E2 -13296.375} C_VEL
LIN {X 0,Y 506.926,Z 293.896,A -85,B 0,C 180,E1 -13298.946,E2 -13298.946} C_VEL
LIN {X 0,Y 506.925,Z 293.893,A -85,B 0,C 180,E1 -13302.303,E2 -13302.303} C_VEL
LIN {X 0,Y 507.002,Z 293.88,A -85,B 0,C 180,E1 -13305.601,E2 -13305.601} C_VEL
LIN {X 0,Y 507.04,Z 293.883,A -85,B 0,C 180,E1 -13308.849,E2 -13308.849} C_VEL
LIN {X 0,Y 507.053,Z 293.875,A -85,B 0,C 180,E1 -13312.06,E2 -13312.06} C_VEL
LIN {X 0,Y 507.165,Z 293.862,A -85,B 0,C 180,E1 -13315.247,E2 -13315.247} C_VEL
LIN {X 0,Y 507.204,Z 293.866,A -85,B 0,C 180,E1 -13319.209,E2 -13319.209} C_VEL
LIN {X 0,Y 507.057,Z 293.868,A -85,B 0,C 180,E1 -13321.583,E2 -13321.583} C_VEL
LIN {X 0,Y 507.174,Z 293.867,A -85,B 0,C 180,E1 -13324.753,E2 -13324.753} C_VEL
LIN {X 0,Y 507.056,Z 293.869,A -85,B 0,C 180,E1 -13327.94,E2 -13327.94} C_VEL
LIN {X 0,Y 507.089,Z 293.869,A -85,B 0,C 180,E1 -13331.282,E2 -13331.282} C_VEL
LIN {X 0,Y 507.018,Z 293.885,A -85,B 0,C 180,E1 -13334.761,E2 -13334.761} C_VEL
LIN {X 0,Y 506.962,Z 293.879,A -85,B 0,C 180,E1 -13337.696,E2 -13337.696} C_VEL
LIN {X 0,Y 506.927,Z 293.891,A -85,B 0,C 180,E1 -13341.054,E2 -13341.054} C_VEL
LIN {X 0,Y 506.892,Z 293.9,A -85,B 0,C 180,E1 -13344.221,E2 -13344.221} C_VEL
LIN {X 0,Y 506.91,Z 293.896,A -85,B 0,C 180,E1 -13347.129,E2 -13347.129} C_VEL
LIN {X 0,Y 506.906,Z 293.896,A -85,B 0,C 180,E1 -13349.831,E2 -13349.831} C_VEL
LIN {X 0,Y 506.93,Z 293.898,A -85,B 0,C 180,E1 -13352.607,E2 -13352.607} C_VEL
LIN {X 0,Y 506.905,Z 293.876,A -85,B 0,C 180,E1 -13355.476,E2 -13355.476} C_VEL
LIN {X 0,Y 506.946,Z 293.891,A -85,B 0,C 180,E1 -13358.046,E2 -13358.046} C_VEL
LIN {X 0,Y 506.926,Z 293.897,A -85,B 0,C 180,E1 -13360.543,E2 -13360.543} C_VEL
LIN {X 0,Y 506.917,Z 293.896,A -85,B 0,C 180,E1 -13363.7,E2 -13363.7} C_VEL
LIN {X 0,Y 506.925,Z 293.894,A -85,B 0,C 180,E1 -13367.082,E2 -13367.082} C_VEL
LIN {X 0,Y 506.926,Z 293.895,A -85,B 0,C 180,E1 -13369.505,E2 -13369.505} C_VEL
LIN {X 0,Y 506.953,Z 293.893,A -85,B 0,C 180,E1 -13372.563,E2 -13372.563} C_VEL
LIN {X 0,Y 506.916,Z 293.906,A -85,B 0,C 180,E1 -13375.495,E2 -13375.495} C_VEL
LIN {X 0,Y 506.914,Z 293.907,A -85,B 0,C 180,E1 -13378.329,E2 -13378.329} C_VEL
LIN {X 0,Y 506.925,Z 294.058,A -85,B 0,C 180,E1 -13380.384,E2 -13380.384} C_VEL
LIN {X 0,Y 510.199,Z 308.023,A -85,B 0,C 180,E1 -13382.842,E2 -13382.842} C_VEL
LIN {X 0,Y 512.272,Z 318.762,A -85,B 0,C 180,E1 -13384.645,E2 -13384.645} C_VEL
LIN {X 0,Y 510.874,Z 335.944,A -85,B 0,C 180,E1 -13387.226,E2 -13387.226} C_VEL
LIN {X 0,Y 509.243,Z 357.514,A -85,B 0,C 180,E1 -13390.414,E2 -13390.414} C_VEL
LIN {X 0,Y 513.914,Z 385.233,A -85,B 0,C 180,E1 -13391.043,E2 -13391.043} C_VEL
LIN {X 0,Y 515.204,Z 396.839,A -85,B 0,C 180,E1 -13391.271,E2 -13391.271} C_VEL
LIN {X 0,Y 513.78,Z 496.164,A -85,B 0,C 180,E1 -13392.696,E2 -13392.696} C_VEL
LIN {X 0,Y 513.131,Z 510.501,A -85,B 0,C 180,E1 -13393.054,E2 -13393.054} C_VEL
LIN {X 0,Y 512.361,Z 523.477,A -85,B 0,C 180,E1 -13393.523,E2 -13393.523} C_VEL
LIN {X 0,Y 511.45,Z 535.746,A -85,B 0,C 180,E1 -13394.105,E2 -13394.105} C_VEL
LIN {X 0,Y 510.386,Z 548.625,A -85,B 0,C 180,E1 -13394.888,E2 -13394.888} C_VEL
LIN {X 0,Y 509.372,Z 560.345,A -85,B 0,C 180,E1 -13395.773,E2 -13395.773} C_VEL
LIN {X 0,Y 508.3,Z 572.074,A -85,B 0,C 180,E1 -13396.86,E2 -13396.86} C_VEL
LIN {X 0,Y 507.463,Z 582.59,A -85,B 0,C 180,E1 -13398.053,E2 -13398.053} C_VEL
LIN {X 0,Y 506.753,Z 591.36,A -85,B 0,C 180,E1 -13399.257,E2 -13399.257} C_VEL
LIN {X 0,Y 506.102,Z 599.692,A -85,B 0,C 180,E1 -13400.643,E2 -13400.643} C_VEL
LIN {X 0,Y 505.607,Z 606.468,A -85,B 0,C 180,E1 -13402.039,E2 -13402.039} C_VEL
LIN {X 0,Y 505.368,Z 616.165,A -85,B 0,C 180,E1 -13404.434,E2 -13404.434} C_VEL
LIN {X 0,Y 505.286,Z 620.04,A -85,B 0,C 180,E1 -13405.629,E2 -13405.629} C_VEL
LIN {X 0,Y 505.274,Z 623.014,A -85,B 0,C 180,E1 -13406.823,E2 -13406.823} C_VEL
LIN {X 0,Y 505.316,Z 625.597,A -85,B 0,C 180,E1 -13408.413,E2 -13408.413} C_VEL
LIN {X 0,Y 505.331,Z 626.714,A -85,B 0,C 180,E1 -13410.002,E2 -13410.002} C_VEL
LIN {X 0,Y 505.297,Z 626.391,A -85,B 0,C 180,E1 -13411.591,E2 -13411.591} C_VEL
LIN {X 0,Y 505.276,Z 624.64,A -85,B 0,C 180,E1 -13413.181,E2 -13413.181} C_VEL
LIN {X 0,Y 505.339,Z 621.43,A -85,B 0,C 180,E1 -13414.772,E2 -13414.772} C_VEL
LIN {X 0,Y 505.418,Z 617.98,A -85,B 0,C 180,E1 -13415.968,E2 -13415.968} C_VEL
LIN {X 0,Y 505.677,Z 611.947,A -85,B 0,C 180,E1 -13417.563,E2 -13417.563} C_VEL
LIN {X 0,Y 506.062,Z 605.153,A -85,B 0,C 180,E1 -13418.96,E2 -13418.96} C_VEL
LIN {X 0,Y 506.695,Z 596.663,A -85,B 0,C 180,E1 -13420.355,E2 -13420.355} C_VEL
LIN {X 0,Y 507.334,Z 588.124,A -85,B 0,C 180,E1 -13421.51,E2 -13421.51} C_VEL
LIN {X 0,Y 508.134,Z 577.056,A -85,B 0,C 180,E1 -13422.743,E2 -13422.743} C_VEL
LIN {X 0,Y 508.967,Z 566.271,A -85,B 0,C 180,E1 -13423.735,E2 -13423.735} C_VEL
LIN {X 0,Y 509.844,Z 554.541,A -85,B 0,C 180,E1 -13424.624,E2 -13424.624} C_VEL
LIN {X 0,Y 510.623,Z 543.444,A -85,B 0,C 180,E1 -13425.313,E2 -13425.313} C_VEL
LIN {X 0,Y 511.447,Z 529.62,A -85,B 0,C 180,E1 -13426.001,E2 -13426.001} C_VEL
LIN {X 0,Y 512.194,Z 515.91,A -85,B 0,C 180,E1 -13426.512,E2 -13426.512} C_VEL
LIN {X 0,Y 512.789,Z 500.686,A -85,B 0,C 180,E1 -13426.902,E2 -13426.902} C_VEL
LIN {X 0,Y 515.498,Z 396.471,A -85,B 0,C 180,E1 -13428.778,E2 -13428.778} C_VEL
LIN {X 0,Y 513.414,Z 376.251,A -85,B 0,C 180,E1 -13429.298,E2 -13429.298} C_VEL
LIN {X 0,Y 510.105,Z 355.07,A -85,B 0,C 180,E1 -13429.924,E2 -13429.924} C_VEL
LIN {X 0,Y 508.764,Z 343.931,A -85,B 0,C 180,E1 -13430.485,E2 -13430.485} C_VEL
LIN {X 0,Y 510.035,Z 323.164,A -85,B 0,C 180,E1 -13433.471,E2 -13433.471} C_VEL
LIN {X 0,Y 510.667,Z 312.814,A -85,B 0,C 180,E1 -13434.978,E2 -13434.978} C_VEL
LIN {X 0,Y 506.963,Z 293.892,A -85,B 0,C 180,E1 -13437.989,E2 -13437.989} C_VEL
LIN {X 0,Y 506.89,Z 293.902,A -85,B 0,C 180,E1 -13441.047,E2 -13441.047} C_VEL
LIN {X 0,Y 506.884,Z 293.903,A -85,B 0,C 180,E1 -13444.513,E2 -13444.513} C_VEL
LIN {X 0,Y 506.854,Z 293.91,A -85,B 0,C 180,E1 -13447.451,E2 -13447.451} C_VEL
LIN {X 0,Y 506.873,Z 293.903,A -85,B 0,C 180,E1 -13450.532,E2 -13450.532} C_VEL
LIN {X 0,Y 506.911,Z 293.898,A -85,B 0,C 180,E1 -13453.703,E2 -13453.703} C_VEL
LIN {X 0,Y 506.923,Z 293.896,A -85,B 0,C 180,E1 -13456.3,E2 -13456.3} C_VEL
LIN {X 0,Y 506.889,Z 293.901,A -85,B 0,C 180,E1 -13459.498,E2 -13459.498} C_VEL
LIN {X 0,Y 506.923,Z 293.901,A -85,B 0,C 180,E1 -13462.557,E2 -13462.557} C_VEL
LIN {X 0,Y 506.899,Z 293.899,A -85,B 0,C 180,E1 -13465.49,E2 -13465.49} C_VEL
LIN {X 0,Y 506.9,Z 293.904,A -85,B 0,C 180,E1 -13468.326,E2 -13468.326} C_VEL
LIN {X 0,Y 506.907,Z 293.899,A -85,B 0,C 180,E1 -13471.077,E2 -13471.077} C_VEL
LIN {X 0,Y 506.904,Z 293.902,A -85,B 0,C 180,E1 -13473.922,E2 -13473.922} C_VEL
LIN {X 0,Y 506.905,Z 293.907,A -85,B 0,C 180,E1 -13476.377,E2 -13476.377} C_VEL
LIN {X 0,Y 506.958,Z 293.901,A -85,B 0,C 180,E1 -13478.947,E2 -13478.947} C_VEL
LIN {X 0,Y 506.957,Z 293.9,A -85,B 0,C 180,E1 -13482.304,E2 -13482.304} C_VEL
LIN {X 0,Y 506.985,Z 293.99,A -85,B 0,C 180,E1 -13484.602,E2 -13484.602} C_VEL
LIN {X 0,Y 510.117,Z 305.456,A -85,B 0,C 180,E1 -13486.501,E2 -13486.501} C_VEL
LIN {X 0,Y 512.598,Z 317.299,A -85,B 0,C 180,E1 -13488.372,E2 -13488.372} C_VEL
LIN {X 0,Y 512.141,Z 331.606,A -85,B 0,C 180,E1 -13490.364,E2 -13490.364} C_VEL
LIN {X 0,Y 511.409,Z 344.731,A -85,B 0,C 180,E1 -13492.165,E2 -13492.165} C_VEL
LIN {X 0,Y 515.917,Z 366.307,A -85,B 0,C 180,E1 -13492.858,E2 -13492.858} C_VEL
LIN {X 0,Y 516.507,Z 371.326,A -85,B 0,C 180,E1 -13492.99,E2 -13492.99} C_VEL
LIN {X 0,Y 513.437,Z 484.553,A -85,B 0,C 180,E1 -13495.031,E2 -13495.031} C_VEL
LIN {X 0,Y 512.954,Z 497.452,A -85,B 0,C 180,E1 -13495.399,E2 -13495.399} C_VEL
LIN {X 0,Y 512.121,Z 512.168,A -85,B 0,C 180,E1 -13495.98,E2 -13495.98} C_VEL
LIN {X 0,Y 511.305,Z 525.185,A -85,B 0,C 180,E1 -13496.662,E2 -13496.662} C_VEL
LIN {X 0,Y 510.347,Z 538.517,A -85,B 0,C 180,E1 -13497.542,E2 -13497.542} C_VEL
LIN {X 0,Y 509.481,Z 550.49,A -85,B 0,C 180,E1 -13498.523,E2 -13498.523} C_VEL
LIN {X 0,Y 508.641,Z 561.299,A -85,B 0,C 180,E1 -13499.605,E2 -13499.605} C_VEL
LIN {X 0,Y 507.67,Z 571.11,A -85,B 0,C 180,E1 -13500.791,E2 -13500.791} C_VEL
LIN {X 0,Y 506.925,Z 580.474,A -85,B 0,C 180,E1 -13502.178,E2 -13502.178} C_VEL
LIN {X 0,Y 506.237,Z 588.088,A -85,B 0,C 180,E1 -13503.57,E2 -13503.57} C_VEL
LIN {X 0,Y 506.032,Z 593.33,A -85,B 0,C 180,E1 -13504.764,E2 -13504.764} C_VEL
LIN {X 0,Y 505.652,Z 598.88,A -85,B 0,C 180,E1 -13506.362,E2 -13506.362} C_VEL
LIN {X 0,Y 505.324,Z 602.819,A -85,B 0,C 180,E1 -13507.968,E2 -13507.968} C_VEL
LIN {X 0,Y 505.272,Z 605.234,A -85,B 0,C 180,E1 -13509.576,E2 -13509.576} C_VEL
LIN {X 0,Y 505.228,Z 605.906,A -85,B 0,C 180,E1 -13510.383,E2 -13510.383} C_VEL
LIN {X 0,Y 505.092,Z 606.168,A -85,B 0,C 180,E1 -13512.006,E2 -13512.006} C_VEL
LIN {X 0,Y 505.193,Z 604.965,A -85,B 0,C 180,E1 -13513.633,E2 -13513.633} C_VEL
LIN {X 0,Y 505.161,Z 603.802,A -85,B 0,C 180,E1 -13514.453,E2 -13514.453} C_VEL
LIN {X 0,Y 505.281,Z 600.249,A -85,B 0,C 180,E1 -13516.096,E2 -13516.096} C_VEL
LIN {X 0,Y 505.404,Z 596.656,A -85,B 0,C 180,E1 -13517.294,E2 -13517.294} C_VEL
LIN {X 0,Y 505.579,Z 591.695,A -85,B 0,C 180,E1 -13518.581,E2 -13518.581} C_VEL
LIN {X 0,Y 505.894,Z 585.284,A -85,B 0,C 180,E1 -13519.916,E2 -13519.916} C_VEL
LIN {X 0,Y 506.291,Z 577.073,A -85,B 0,C 180,E1 -13521.295,E2 -13521.295} C_VEL
LIN {X 0,Y 506.751,Z 567.641,A -85,B 0,C 180,E1 -13522.582,E2 -13522.582} C_VEL
LIN {X 0,Y 507.334,Z 556.583,A -85,B 0,C 180,E1 -13523.818,E2 -13523.818} C_VEL
LIN {X 0,Y 508.001,Z 545.115,A -85,B 0,C 180,E1 -13524.869,E2 -13524.869} C_VEL
LIN {X 0,Y 508.643,Z 532.346,A -85,B 0,C 180,E1 -13525.817,E2 -13525.817} C_VEL
LIN {X 0,Y 509.304,Z 518.717,A -85,B 0,C 180,E1 -13526.625,E2 -13526.625} C_VEL
LIN {X 0,Y 509.833,Z 505.488,A -85,B 0,C 180,E1 -13527.237,E2 -13527.237} C_VEL
LIN {X 0,Y 510.403,Z 491.156,A -85,B 0,C 180,E1 -13527.73,E2 -13527.73} C_VEL
LIN {X 0,Y 510.703,Z 476.185,A -85,B 0,C 180,E1 -13528.074,E2 -13528.074} C_VEL
LIN {X 0,Y 512.444,Z 367.725,A -85,B 0,C 180,E1 -13529.867,E2 -13529.867} C_VEL
LIN {X 0,Y 508.934,Z 343.115,A -85,B 0,C 180,E1 -13530.406,E2 -13530.406} C_VEL
LIN {X 0,Y 509.75,Z 321.993,A -85,B 0,C 180,E1 -13533.342,E2 -13533.342} C_VEL
LIN {X 0,Y 510.068,Z 309.937,A -85,B 0,C 180,E1 -13535.025,E2 -13535.025} C_VEL
LIN {X 0,Y 506.969,Z 293.893,A -85,B 0,C 180,E1 -13537.439,E2 -13537.439} C_VEL
LIN {X 0,Y 506.878,Z 293.905,A -85,B 0,C 180,E1 -13540.531,E2 -13540.531} C_VEL
LIN {X 0,Y 506.935,Z 293.894,A -85,B 0,C 180,E1 -13543.698,E2 -13543.698} C_VEL
LIN {X 0,Y 506.901,Z 293.898,A -85,B 0,C 180,E1 -13547.085,E2 -13547.085} C_VEL
LIN {X 0,Y 506.888,Z 293.9,A -85,B 0,C 180,E1 -13549.497,E2 -13549.497} C_VEL
LIN {X 0,Y 506.851,Z 293.908,A -85,B 0,C 180,E1 -13552.549,E2 -13552.549} C_VEL
LIN {X 0,Y 506.887,Z 293.901,A -85,B 0,C 180,E1 -13555.488,E2 -13555.488} C_VEL
LIN {X 0,Y 506.888,Z 293.904,A -85,B 0,C 180,E1 -13558.323,E2 -13558.323} C_VEL
LIN {X 0,Y 506.903,Z 293.898,A -85,B 0,C 180,E1 -13561.075,E2 -13561.075} C_VEL
LIN {X 0,Y 506.895,Z 293.903,A -85,B 0,C 180,E1 -13563.921,E2 -13563.921} C_VEL
LIN {X 0,Y 506.903,Z 293.902,A -85,B 0,C 180,E1 -13566.375,E2 -13566.375} C_VEL
LIN {X 0,Y 506.955,Z 293.891,A -85,B 0,C 180,E1 -13568.945,E2 -13568.945} C_VEL
LIN {X 0,Y 506.974,Z 293.893,A -85,B 0,C 180,E1 -13572.303,E2 -13572.303} C_VEL
LIN {X 0,Y 507.029,Z 293.885,A -85,B 0,C 180,E1 -13575.6,E2 -13575.6} C_VEL
LIN {X 0,Y 507.068,Z 293.876,A -85,B 0,C 180,E1 -13578.847,E2 -13578.847} C_VEL
LIN {X 0,Y 507.094,Z 293.918,A -85,B 0,C 180,E1 -13581.809,E2 -13581.809} C_VEL
LIN {X 0,Y 508.668,Z 303.361,A -85,B 0,C 180,E1 -13583.692,E2 -13583.692} C_VEL
LIN {X 0,Y 512.931,Z 323.885,A -85,B 0,C 180,E1 -13584.12,E2 -13584.12} C_VEL
LIN {X 0,Y 512.49,Z 359.742,A -85,B 0,C 180,E1 -13584.619,E2 -13584.619} C_VEL
LIN {X 0,Y 511.787,Z 365.581,A -85,B 0,C 180,E1 -13584.682,E2 -13584.682} C_VEL
LIN {X 0,Y 505.928,Z 384.522,A -85,B 0,C 180,E1 -13584.782,E2 -13584.782} C_VEL
LIN {X 0,Y 505.203,Z 390.362,A -85,B 0,C 180,E1 -13584.845,E2 -13584.845} C_VEL
LIN {X 0,Y 504.657,Z 439.775,A -85,B 0,C 180,E1 -13585.57,E2 -13585.57} C_VEL
LIN {X 0,Y 504.334,Z 454.024,A -85,B 0,C 180,E1 -13585.941,E2 -13585.941} C_VEL
LIN {X 0,Y 503.832,Z 467.776,A -85,B 0,C 180,E1 -13586.461,E2 -13586.461} C_VEL
LIN {X 0,Y 503.321,Z 480.57,A -85,B 0,C 180,E1 -13587.106,E2 -13587.106} C_VEL
LIN {X 0,Y 502.745,Z 493.002,A -85,B 0,C 180,E1 -13587.902,E2 -13587.902} C_VEL
LIN {X 0,Y 501.864,Z 504.437,A -85,B 0,C 180,E1 -13588.798,E2 -13588.798} C_VEL
LIN {X 0,Y 501.368,Z 514.847,A -85,B 0,C 180,E1 -13589.798,E2 -13589.798} C_VEL
LIN {X 0,Y 500.542,Z 525.268,A -85,B 0,C 180,E1 -13591,E2 -13591} C_VEL
LIN {X 0,Y 499.981,Z 533.85,A -85,B 0,C 180,E1 -13592.206,E2 -13592.206} C_VEL
LIN {X 0,Y 499.423,Z 541.007,A -85,B 0,C 180,E1 -13593.415,E2 -13593.415} C_VEL
LIN {X 0,Y 499.169,Z 548.33,A -85,B 0,C 180,E1 -13594.939,E2 -13594.939} C_VEL
LIN {X 0,Y 498.809,Z 553.995,A -85,B 0,C 180,E1 -13596.448,E2 -13596.448} C_VEL
LIN {X 0,Y 498.496,Z 558.513,A -85,B 0,C 180,E1 -13598.075,E2 -13598.075} C_VEL
LIN {X 0,Y 498.408,Z 561.571,A -85,B 0,C 180,E1 -13599.707,E2 -13599.707} C_VEL
LIN {X 0,Y 498.342,Z 563.265,A -85,B 0,C 180,E1 -13601.346,E2 -13601.346} C_VEL
LIN {X 0,Y 498.373,Z 563.611,A -85,B 0,C 180,E1 -13602.993,E2 -13602.993} C_VEL
LIN {X 0,Y 498.549,Z 562.597,A -85,B 0,C 180,E1 -13604.647,E2 -13604.647} C_VEL
LIN {X 0,Y 498.719,Z 560.194,A -85,B 0,C 180,E1 -13606.311,E2 -13606.311} C_VEL
LIN {X 0,Y 498.98,Z 557.962,A -85,B 0,C 180,E1 -13607.34,E2 -13607.34} C_VEL
LIN {X 0,Y 499.403,Z 553.728,A -85,B 0,C 180,E1 -13608.817,E2 -13608.817} C_VEL
LIN {X 0,Y 499.912,Z 548.759,A -85,B 0,C 180,E1 -13610.156,E2 -13610.156} C_VEL
LIN {X 0,Y 500.537,Z 542.276,A -85,B 0,C 180,E1 -13611.549,E2 -13611.549} C_VEL
LIN {X 0,Y 501.257,Z 535.493,A -85,B 0,C 180,E1 -13612.74,E2 -13612.74} C_VEL
LIN {X 0,Y 502.224,Z 526.312,A -85,B 0,C 180,E1 -13614.073,E2 -13614.073} C_VEL
LIN {X 0,Y 503.231,Z 515.877,A -85,B 0,C 180,E1 -13615.306,E2 -13615.306} C_VEL
LIN {X 0,Y 504.246,Z 504.678,A -85,B 0,C 180,E1 -13616.389,E2 -13616.389} C_VEL
LIN {X 0,Y 505.283,Z 492.181,A -85,B 0,C 180,E1 -13617.37,E2 -13617.37} C_VEL
LIN {X 0,Y 506.148,Z 479.309,A -85,B 0,C 180,E1 -13618.177,E2 -13618.177} C_VEL
LIN {X 0,Y 506.824,Z 466.371,A -85,B 0,C 180,E1 -13618.812,E2 -13618.812} C_VEL
LIN {X 0,Y 507.454,Z 452.492,A -85,B 0,C 180,E1 -13619.316,E2 -13619.316} C_VEL
LIN {X 0,Y 507.825,Z 438.317,A -85,B 0,C 180,E1 -13619.662,E2 -13619.662} C_VEL
LIN {X 0,Y 509.442,Z 326.774,A -85,B 0,C 180,E1 -13621.277,E2 -13621.277} C_VEL
LIN {X 0,Y 506.825,Z 316.984,A -85,B 0,C 180,E1 -13621.551,E2 -13621.551} C_VEL
LIN {X 0,Y 501.849,Z 304.359,A -85,B 0,C 180,E1 -13622.007,E2 -13622.007} C_VEL
LIN {X 0,Y 499.816,Z 294.786,A -85,B 0,C 180,E1 -13624.157,E2 -13624.157} C_VEL
LIN {X 0,Y 499.865,Z 294.776,A -85,B 0,C 180,E1 -13627.049,E2 -13627.049} C_VEL
LIN {X 0,Y 499.81,Z 294.789,A -85,B 0,C 180,E1 -13630.136,E2 -13630.136} C_VEL
LIN {X 0,Y 499.862,Z 294.779,A -85,B 0,C 180,E1 -13633.36,E2 -13633.36} C_VEL
LIN {X 0,Y 499.861,Z 294.776,A -85,B 0,C 180,E1 -13636.771,E2 -13636.771} C_VEL
LIN {X 0,Y 499.814,Z 294.784,A -85,B 0,C 180,E1 -13639.861,E2 -13639.861} C_VEL
LIN {X 0,Y 499.873,Z 294.77,A -85,B 0,C 180,E1 -13643.002,E2 -13643.002} C_VEL
LIN {X 0,Y 499.828,Z 294.774,A -85,B 0,C 180,E1 -13645.906,E2 -13645.906} C_VEL
LIN {X 0,Y 499.857,Z 294.771,A -85,B 0,C 180,E1 -13648.77,E2 -13648.77} C_VEL
LIN {X 0,Y 499.879,Z 294.77,A -85,B 0,C 180,E1 -13651.973,E2 -13651.973} C_VEL
LIN {X 0,Y 499.815,Z 294.782,A -85,B 0,C 180,E1 -13654.251,E2 -13654.251} C_VEL
LIN {X 0,Y 499.837,Z 294.771,A -85,B 0,C 180,E1 -13656.898,E2 -13656.898} C_VEL
LIN {X 0,Y 499.898,Z 294.769,A -85,B 0,C 180,E1 -13659.841,E2 -13659.841} C_VEL
LIN {X 0,Y 499.887,Z 294.771,A -85,B 0,C 180,E1 -13662.887,E2 -13662.887} C_VEL
LIN {X 0,Y 499.952,Z 294.759,A -85,B 0,C 180,E1 -13665.393,E2 -13665.393} C_VEL
LIN {X 0,Y 499.996,Z 294.759,A -85,B 0,C 180,E1 -13668.69,E2 -13668.69} C_VEL
LIN {X 0,Y 500.01,Z 294.753,A -85,B 0,C 180,E1 -13671.947,E2 -13671.947} C_VEL
LIN {X 0,Y 500.042,Z 294.752,A -85,B 0,C 180,E1 -13674.373,E2 -13674.373} C_VEL
LIN {X 0,Y 499.995,Z 294.749,A -85,B 0,C 180,E1 -13676.788,E2 -13676.788} C_VEL
LIN {X 0,Y 500.167,Z 294.735,A -85,B 0,C 180,E1 -13680,E2 -13680} C_VEL
LIN {X 0,Y 500.088,Z 294.745,A -85,B 0,C 180,E1 -13684.016,E2 -13684.016} C_VEL
LIN {X 0,Y 500.057,Z 294.748,A -85,B 0,C 180,E1 -13686.434,E2 -13686.434} C_VEL
LIN {X 0,Y 499.978,Z 294.758,A -85,B 0,C 180,E1 -13688.865,E2 -13688.865} C_VEL
LIN {X 0,Y 500.047,Z 294.745,A -85,B 0,C 180,E1 -13691.339,E2 -13691.339} C_VEL
LIN {X 0,Y 499.981,Z 294.764,A -85,B 0,C 180,E1 -13694.85,E2 -13694.85} C_VEL
LIN {X 0,Y 499.914,Z 294.757,A -85,B 0,C 180,E1 -13697.954,E2 -13697.954} C_VEL
LIN {X 0,Y 499.883,Z 294.776,A -85,B 0,C 180,E1 -13700.506,E2 -13700.506} C_VEL
LIN {X 0,Y 499.837,Z 294.779,A -85,B 0,C 180,E1 -13703.103,E2 -13703.103} C_VEL
LIN {X 0,Y 499.88,Z 294.771,A -85,B 0,C 180,E1 -13706.268,E2 -13706.268} C_VEL
LIN {X 0,Y 499.871,Z 294.772,A -85,B 0,C 180,E1 -13709.369,E2 -13709.369} C_VEL
LIN {X 0,Y 499.894,Z 294.773,A -85,B 0,C 180,E1 -13712.171,E2 -13712.171} C_VEL
LIN {X 0,Y 499.865,Z 294.753,A -85,B 0,C 180,E1 -13715.066,E2 -13715.066} C_VEL
LIN {X 0,Y 499.898,Z 294.769,A -85,B 0,C 180,E1 -13718.062,E2 -13718.062} C_VEL
LIN {X 0,Y 499.878,Z 294.775,A -85,B 0,C 180,E1 -13720.833,E2 -13720.833} C_VEL
LIN {X 0,Y 499.866,Z 294.773,A -85,B 0,C 180,E1 -13723.363,E2 -13723.363} C_VEL
LIN {X 0,Y 499.872,Z 294.775,A -85,B 0,C 180,E1 -13726.641,E2 -13726.641} C_VEL
LIN {X 0,Y 499.884,Z 294.771,A -85,B 0,C 180,E1 -13729.17,E2 -13729.17} C_VEL
LIN {X 0,Y 499.902,Z 294.776,A -85,B 0,C 180,E1 -13731.941,E2 -13731.941} C_VEL
LIN {X 0,Y 499.872,Z 294.781,A -85,B 0,C 180,E1 -13734.938,E2 -13734.938} C_VEL
LIN {X 0,Y 499.891,Z 294.783,A -85,B 0,C 180,E1 -13737.832,E2 -13737.832} C_VEL
LIN {X 0,Y 499.858,Z 294.828,A -85,B 0,C 180,E1 -13740.051,E2 -13740.051} C_VEL
LIN {X 0,Y 502.98,Z 307.996,A -85,B 0,C 180,E1 -13742.42,E2 -13742.42} C_VEL
LIN {X 0,Y 505.26,Z 318.947,A -85,B 0,C 180,E1 -13744.303,E2 -13744.303} C_VEL
LIN {X 0,Y 505.223,Z 323.291,A -85,B 0,C 180,E1 -13744.988,E2 -13744.988} C_VEL
LIN {X 0,Y 503.691,Z 339.96,A -85,B 0,C 180,E1 -13747.519,E2 -13747.519} C_VEL
LIN {X 0,Y 502.413,Z 357.079,A -85,B 0,C 180,E1 -13750.086,E2 -13750.086} C_VEL
LIN {X 0,Y 507.215,Z 385.503,A -85,B 0,C 180,E1 -13750.745,E2 -13750.745} C_VEL
LIN {X 0,Y 508.613,Z 397.724,A -85,B 0,C 180,E1 -13750.992,E2 -13750.992} C_VEL
LIN {X 0,Y 507.138,Z 495.746,A -85,B 0,C 180,E1 -13752.416,E2 -13752.416} C_VEL
LIN {X 0,Y 506.451,Z 510.343,A -85,B 0,C 180,E1 -13752.786,E2 -13752.786} C_VEL
LIN {X 0,Y 505.667,Z 522.935,A -85,B 0,C 180,E1 -13753.247,E2 -13753.247} C_VEL
LIN {X 0,Y 504.64,Z 536.108,A -85,B 0,C 180,E1 -13753.885,E2 -13753.885} C_VEL
LIN {X 0,Y 503.548,Z 548.835,A -85,B 0,C 180,E1 -13754.677,E2 -13754.677} C_VEL
LIN {X 0,Y 502.389,Z 561.603,A -85,B 0,C 180,E1 -13755.674,E2 -13755.674} C_VEL
LIN {X 0,Y 501.363,Z 572.07,A -85,B 0,C 180,E1 -13756.675,E2 -13756.675} C_VEL
LIN {X 0,Y 500.477,Z 582.507,A -85,B 0,C 180,E1 -13757.884,E2 -13757.884} C_VEL
LIN {X 0,Y 499.716,Z 591.596,A -85,B 0,C 180,E1 -13759.161,E2 -13759.161} C_VEL
LIN {X 0,Y 499.076,Z 599.493,A -85,B 0,C 180,E1 -13760.51,E2 -13760.51} C_VEL
LIN {X 0,Y 498.537,Z 606.223,A -85,B 0,C 180,E1 -13761.925,E2 -13761.925} C_VEL
LIN {X 0,Y 498.275,Z 615.774,A -85,B 0,C 180,E1 -13764.355,E2 -13764.355} C_VEL
LIN {X 0,Y 498.199,Z 619.712,A -85,B 0,C 180,E1 -13765.567,E2 -13765.567} C_VEL
LIN {X 0,Y 498.192,Z 622.72,A -85,B 0,C 180,E1 -13766.778,E2 -13766.778} C_VEL
LIN {X 0,Y 498.232,Z 625.381,A -85,B 0,C 180,E1 -13768.391,E2 -13768.391} C_VEL
LIN {X 0,Y 498.24,Z 626.549,A -85,B 0,C 180,E1 -13770.002,E2 -13770.002} C_VEL
LIN {X 0,Y 498.213,Z 626.277,A -85,B 0,C 180,E1 -13771.613,E2 -13771.613} C_VEL
LIN {X 0,Y 498.194,Z 624.57,A -85,B 0,C 180,E1 -13773.226,E2 -13773.226} C_VEL
LIN {X 0,Y 498.252,Z 621.404,A -85,B 0,C 180,E1 -13774.84,E2 -13774.84} C_VEL
LIN {X 0,Y 498.395,Z 616.703,A -85,B 0,C 180,E1 -13776.457,E2 -13776.457} C_VEL
LIN {X 0,Y 498.628,Z 612.031,A -85,B 0,C 180,E1 -13777.671,E2 -13777.671} C_VEL
LIN {X 0,Y 499.051,Z 605.286,A -85,B 0,C 180,E1 -13779.087,E2 -13779.087} C_VEL
LIN {X 0,Y 499.698,Z 596.888,A -85,B 0,C 180,E1 -13780.501,E2 -13780.501} C_VEL
LIN {X 0,Y 500.365,Z 588.437,A -85,B 0,C 180,E1 -13781.672,E2 -13781.672} C_VEL
LIN {X 0,Y 501.228,Z 577.479,A -85,B 0,C 180,E1 -13782.922,E2 -13782.922} C_VEL
LIN {X 0,Y 502.144,Z 565.619,A -85,B 0,C 180,E1 -13784.028,E2 -13784.028} C_VEL
LIN {X 0,Y 503.144,Z 553.805,A -85,B 0,C 180,E1 -13784.926,E2 -13784.926} C_VEL
LIN {X 0,Y 503.818,Z 544.347,A -85,B 0,C 180,E1 -13785.525,E2 -13785.525} C_VEL
LIN {X 0,Y 504.707,Z 530.85,A -85,B 0,C 180,E1 -13786.22,E2 -13786.22} C_VEL
LIN {X 0,Y 505.483,Z 516.958,A -85,B 0,C 180,E1 -13786.764,E2 -13786.764} C_VEL
LIN {X 0,Y 506.169,Z 502.374,A -85,B 0,C 180,E1 -13787.161,E2 -13787.161} C_VEL
LIN {X 0,Y 509.034,Z 396.535,A -85,B 0,C 180,E1 -13789.118,E2 -13789.118} C_VEL
LIN {X 0,Y 506.98,Z 376.806,A -85,B 0,C 180,E1 -13789.645,E2 -13789.645} C_VEL
LIN {X 0,Y 503.575,Z 355.307,A -85,B 0,C 180,E1 -13790.305,E2 -13790.305} C_VEL
LIN {X 0,Y 501.946,Z 341.76,A -85,B 0,C 180,E1 -13790.991,E2 -13790.991} C_VEL
LIN {X 0,Y 503.46,Z 319.571,A -85,B 0,C 180,E1 -13794.233,E2 -13794.233} C_VEL
LIN {X 0,Y 503.717,Z 314.368,A -85,B 0,C 180,E1 -13795.002,E2 -13795.002} C_VEL
LIN {X 0,Y 500.034,Z 295.326,A -85,B 0,C 180,E1 -13798.054,E2 -13798.054} C_VEL
LIN {X 0,Y 499.907,Z 294.77,A -85,B 0,C 180,E1 -13798.202,E2 -13798.202} C_VEL
LIN {X 0,Y 499.838,Z 294.782,A -85,B 0,C 180,E1 -13801.26,E2 -13801.26} C_VEL
LIN {X 0,Y 499.848,Z 294.78,A -85,B 0,C 180,E1 -13804.231,E2 -13804.231} C_VEL
LIN {X 0,Y 499.833,Z 294.781,A -85,B 0,C 180,E1 -13807.057,E2 -13807.057} C_VEL
LIN {X 0,Y 499.832,Z 294.781,A -85,B 0,C 180,E1 -13810.139,E2 -13810.139} C_VEL
LIN {X 0,Y 499.867,Z 294.777,A -85,B 0,C 180,E1 -13813.365,E2 -13813.365} C_VEL
LIN {X 0,Y 499.87,Z 294.776,A -85,B 0,C 180,E1 -13816.775,E2 -13816.775} C_VEL
LIN {X 0,Y 499.832,Z 294.779,A -85,B 0,C 180,E1 -13819.862,E2 -13819.862} C_VEL
LIN {X 0,Y 499.895,Z 294.775,A -85,B 0,C 180,E1 -13823.006,E2 -13823.006} C_VEL
LIN {X 0,Y 499.854,Z 294.777,A -85,B 0,C 180,E1 -13825.908,E2 -13825.908} C_VEL
LIN {X 0,Y 499.887,Z 294.776,A -85,B 0,C 180,E1 -13828.772,E2 -13828.772} C_VEL
LIN {X 0,Y 499.902,Z 294.773,A -85,B 0,C 180,E1 -13831.976,E2 -13831.976} C_VEL
LIN {X 0,Y 499.852,Z 294.781,A -85,B 0,C 180,E1 -13835.141,E2 -13835.141} C_VEL
LIN {X 0,Y 499.927,Z 294.777,A -85,B 0,C 180,E1 -13837.772,E2 -13837.772} C_VEL
LIN {X 0,Y 499.927,Z 294.781,A -85,B 0,C 180,E1 -13840.351,E2 -13840.351} C_VEL
LIN {X 0,Y 499.912,Z 294.774,A -85,B 0,C 180,E1 -13842.888,E2 -13842.888} C_VEL
LIN {X 0,Y 499.91,Z 294.788,A -85,B 0,C 180,E1 -13844.144,E2 -13844.144} C_VEL
LIN {X 0,Y 503.193,Z 306.351,A -85,B 0,C 180,E1 -13846.106,E2 -13846.106} C_VEL
LIN {X 0,Y 505.739,Z 318.138,A -85,B 0,C 180,E1 -13848.01,E2 -13848.01} C_VEL
LIN {X 0,Y 505.985,Z 322.293,A -85,B 0,C 180,E1 -13848.623,E2 -13848.623} C_VEL
LIN {X 0,Y 505.027,Z 340.79,A -85,B 0,C 180,E1 -13851.224,E2 -13851.224} C_VEL
LIN {X 0,Y 504.792,Z 344.75,A -85,B 0,C 180,E1 -13851.773,E2 -13851.773} C_VEL
LIN {X 0,Y 509.384,Z 366.761,A -85,B 0,C 180,E1 -13852.506,E2 -13852.506} C_VEL
LIN {X 0,Y 510.112,Z 371.917,A -85,B 0,C 180,E1 -13852.653,E2 -13852.653} C_VEL
LIN {X 0,Y 506.843,Z 484.867,A -85,B 0,C 180,E1 -13854.737,E2 -13854.737} C_VEL
LIN {X 0,Y 506.284,Z 498.801,A -85,B 0,C 180,E1 -13855.149,E2 -13855.149} C_VEL
LIN {X 0,Y 505.397,Z 513.451,A -85,B 0,C 180,E1 -13855.753,E2 -13855.753} C_VEL
LIN {X 0,Y 504.6,Z 525.832,A -85,B 0,C 180,E1 -13856.419,E2 -13856.419} C_VEL
LIN {X 0,Y 503.57,Z 539.069,A -85,B 0,C 180,E1 -13857.309,E2 -13857.309} C_VEL
LIN {X 0,Y 502.658,Z 550.948,A -85,B 0,C 180,E1 -13858.303,E2 -13858.303} C_VEL
LIN {X 0,Y 501.768,Z 561.692,A -85,B 0,C 180,E1 -13859.4,E2 -13859.4} C_VEL
LIN {X 0,Y 500.758,Z 571.477,A -85,B 0,C 180,E1 -13860.601,E2 -13860.601} C_VEL
LIN {X 0,Y 500.065,Z 579.589,A -85,B 0,C 180,E1 -13861.806,E2 -13861.806} C_VEL
LIN {X 0,Y 499.316,Z 587.381,A -85,B 0,C 180,E1 -13863.217,E2 -13863.217} C_VEL
LIN {X 0,Y 498.973,Z 593.72,A -85,B 0,C 180,E1 -13864.659,E2 -13864.659} C_VEL
LIN {X 0,Y 498.645,Z 598.507,A -85,B 0,C 180,E1 -13866.047,E2 -13866.047} C_VEL
LIN {X 0,Y 498.379,Z 601.73,A -85,B 0,C 180,E1 -13867.267,E2 -13867.267} C_VEL
LIN {X 0,Y 498.204,Z 604.686,A -85,B 0,C 180,E1 -13868.897,E2 -13868.897} C_VEL
LIN {X 0,Y 498.132,Z 606.196,A -85,B 0,C 180,E1 -13870.533,E2 -13870.533} C_VEL
LIN {X 0,Y 497.995,Z 606.264,A -85,B 0,C 180,E1 -13872.18,E2 -13872.18} C_VEL
LIN {X 0,Y 498.094,Z 604.812,A -85,B 0,C 180,E1 -13873.831,E2 -13873.831} C_VEL
LIN {X 0,Y 498.107,Z 601.821,A -85,B 0,C 180,E1 -13875.497,E2 -13875.497} C_VEL
LIN {X 0,Y 498.271,Z 597.514,A -85,B 0,C 180,E1 -13877.074,E2 -13877.074} C_VEL
LIN {X 0,Y 498.466,Z 592.538,A -85,B 0,C 180,E1 -13878.431,E2 -13878.431} C_VEL
LIN {X 0,Y 498.788,Z 586.221,A -85,B 0,C 180,E1 -13879.798,E2 -13879.798} C_VEL
LIN {X 0,Y 499.137,Z 578.297,A -85,B 0,C 180,E1 -13881.183,E2 -13881.183} C_VEL
LIN {X 0,Y 499.625,Z 569.524,A -85,B 0,C 180,E1 -13882.437,E2 -13882.437} C_VEL
LIN {X 0,Y 500.193,Z 559.38,A -85,B 0,C 180,E1 -13883.631,E2 -13883.631} C_VEL
LIN {X 0,Y 500.76,Z 548.885,A -85,B 0,C 180,E1 -13884.657,E2 -13884.657} C_VEL
LIN {X 0,Y 501.461,Z 536.406,A -85,B 0,C 180,E1 -13885.659,E2 -13885.659} C_VEL
LIN {X 0,Y 502.088,Z 523.218,A -85,B 0,C 180,E1 -13886.514,E2 -13886.514} C_VEL
LIN {X 0,Y 502.701,Z 509.559,A -85,B 0,C 180,E1 -13887.209,E2 -13887.209} C_VEL
LIN {X 0,Y 503.254,Z 494.906,A -85,B 0,C 180,E1 -13887.764,E2 -13887.764} C_VEL
LIN {X 0,Y 503.707,Z 479.659,A -85,B 0,C 180,E1 -13888.159,E2 -13888.159} C_VEL
LIN {X 0,Y 505.548,Z 368.388,A -85,B 0,C 180,E1 -13890.046,E2 -13890.046} C_VEL
LIN {X 0,Y 501.98,Z 343.263,A -85,B 0,C 180,E1 -13890.602,E2 -13890.602} C_VEL
LIN {X 0,Y 502.815,Z 322.384,A -85,B 0,C 180,E1 -13893.525,E2 -13893.525} C_VEL
LIN {X 0,Y 503.157,Z 311.552,A -85,B 0,C 180,E1 -13895.047,E2 -13895.047} C_VEL
LIN {X 0,Y 499.922,Z 294.771,A -85,B 0,C 180,E1 -13897.583,E2 -13897.583} C_VEL
LIN {X 0,Y 499.825,Z 294.782,A -85,B 0,C 180,E1 -13900.82,E2 -13900.82} C_VEL
LIN {X 0,Y 499.886,Z 294.771,A -85,B 0,C 180,E1 -13903.361,E2 -13903.361} C_VEL
LIN {X 0,Y 499.87,Z 294.776,A -85,B 0,C 180,E1 -13906.773,E2 -13906.773} C_VEL
LIN {X 0,Y 499.831,Z 294.782,A -85,B 0,C 180,E1 -13909.861,E2 -13909.861} C_VEL
LIN {X 0,Y 499.837,Z 294.779,A -85,B 0,C 180,E1 -13913.013,E2 -13913.013} C_VEL
LIN {X 0,Y 499.846,Z 294.782,A -85,B 0,C 180,E1 -13915.906,E2 -13915.906} C_VEL
LIN {X 0,Y 499.843,Z 294.779,A -85,B 0,C 180,E1 -13918.767,E2 -13918.767} C_VEL
LIN {X 0,Y 499.842,Z 294.779,A -85,B 0,C 180,E1 -13921.544,E2 -13921.544} C_VEL
LIN {X 0,Y 499.834,Z 294.784,A -85,B 0,C 180,E1 -13924.25,E2 -13924.25} C_VEL
LIN {X 0,Y 499.865,Z 294.775,A -85,B 0,C 180,E1 -13926.897,E2 -13926.897} C_VEL
LIN {X 0,Y 499.926,Z 294.771,A -85,B 0,C 180,E1 -13929.84,E2 -13929.84} C_VEL
LIN {X 0,Y 499.926,Z 294.766,A -85,B 0,C 180,E1 -13932.887,E2 -13932.887} C_VEL
LIN {X 0,Y 499.98,Z 294.762,A -85,B 0,C 180,E1 -13935.392,E2 -13935.392} C_VEL
LIN {X 0,Y 500.044,Z 294.751,A -85,B 0,C 180,E1 -13938.689,E2 -13938.689} C_VEL
LIN {X 0,Y 500.092,Z 294.944,A -85,B 0,C 180,E1 -13941.693,E2 -13941.693} C_VEL
LIN {X 0,Y 501.586,Z 303.581,A -85,B 0,C 180,E1 -13943.464,E2 -13943.464} C_VEL
LIN {X 0,Y 504.528,Z 317.215,A -85,B 0,C 180,E1 -13943.762,E2 -13943.762} C_VEL
LIN {X 0,Y 506.171,Z 326.011,A -85,B 0,C 180,E1 -13943.941,E2 -13943.941} C_VEL
LIN {X 0,Y 505.203,Z 390.362,A -85,B 0,C 180,E1 -13944.845,E2 -13944.845} C_VEL
LIN {X 0,Y 504.461,Z 396.208,A -85,B 0,C 180,E1 -13944.908,E2 -13944.908} C_VEL
LIN {X 0,Y 498.578,Z 415.156,A -85,B 0,C 180,E1 -13945.013,E2 -13945.013} C_VEL
LIN {X 0,Y 497.98,Z 420.995,A -85,B 0,C 180,E1 -13945.081,E2 -13945.081} C_VEL
LIN {X 0,Y 497.742,Z 441.308,A -85,B 0,C 180,E1 -13945.407,E2 -13945.407} C_VEL
LIN {X 0,Y 497.429,Z 455.911,A -85,B 0,C 180,E1 -13945.809,E2 -13945.809} C_VEL
LIN {X 0,Y 496.865,Z 469.849,A -85,B 0,C 180,E1 -13946.361,E2 -13946.361} C_VEL
LIN {X 0,Y 496.303,Z 483.151,A -85,B 0,C 180,E1 -13947.066,E2 -13947.066} C_VEL
LIN {X 0,Y 495.615,Z 495.198,A -85,B 0,C 180,E1 -13947.872,E2 -13947.872} C_VEL
LIN {X 0,Y 494.737,Z 507.401,A -85,B 0,C 180,E1 -13948.883,E2 -13948.883} C_VEL
LIN {X 0,Y 494.173,Z 518.281,A -85,B 0,C 180,E1 -13949.998,E2 -13949.998} C_VEL
LIN {X 0,Y 493.357,Z 528.143,A -85,B 0,C 180,E1 -13951.218,E2 -13951.218} C_VEL
LIN {X 0,Y 492.833,Z 536.31,A -85,B 0,C 180,E1 -13952.442,E2 -13952.442} C_VEL
LIN {X 0,Y 492.264,Z 543.156,A -85,B 0,C 180,E1 -13953.669,E2 -13953.669} C_VEL
LIN {X 0,Y 492.108,Z 548.811,A -85,B 0,C 180,E1 -13954.897,E2 -13954.897} C_VEL
LIN {X 0,Y 491.777,Z 553.447,A -85,B 0,C 180,E1 -13956.13,E2 -13956.13} C_VEL
LIN {X 0,Y 491.48,Z 558.261,A -85,B 0,C 180,E1 -13957.779,E2 -13957.779} C_VEL
LIN {X 0,Y 491.362,Z 560.86,A -85,B 0,C 180,E1 -13959.019,E2 -13959.019} C_VEL
LIN {X 0,Y 491.286,Z 563.13,A -85,B 0,C 180,E1 -13960.679,E2 -13960.679} C_VEL
LIN {X 0,Y 491.251,Z 564.051,A -85,B 0,C 180,E1 -13962.347,E2 -13962.347} C_VEL
LIN {X 0,Y 491.452,Z 563.614,A -85,B 0,C 180,E1 -13964.02,E2 -13964.02} C_VEL
LIN {X 0,Y 491.551,Z 561.815,A -85,B 0,C 180,E1 -13965.706,E2 -13965.706} C_VEL
LIN {X 0,Y 491.926,Z 558.547,A -85,B 0,C 180,E1 -13967.396,E2 -13967.396} C_VEL
LIN {X 0,Y 492.442,Z 553.692,A -85,B 0,C 180,E1 -13969.093,E2 -13969.093} C_VEL
LIN {X 0,Y 492.995,Z 548.55,A -85,B 0,C 180,E1 -13970.463,E2 -13970.463} C_VEL
LIN {X 0,Y 493.673,Z 541.978,A -85,B 0,C 180,E1 -13971.864,E2 -13971.864} C_VEL
LIN {X 0,Y 494.456,Z 535.016,A -85,B 0,C 180,E1 -13973.083,E2 -13973.083} C_VEL
LIN {X 0,Y 495.443,Z 525.677,A -85,B 0,C 180,E1 -13974.424,E2 -13974.424} C_VEL
LIN {X 0,Y 496.46,Z 515.975,A -85,B 0,C 180,E1 -13975.571,E2 -13975.571} C_VEL
LIN {X 0,Y 497.508,Z 504.786,A -85,B 0,C 180,E1 -13976.662,E2 -13976.662} C_VEL
LIN {X 0,Y 498.543,Z 492.714,A -85,B 0,C 180,E1 -13977.62,E2 -13977.62} C_VEL
LIN {X 0,Y 499.421,Z 480.257,A -85,B 0,C 180,E1 -13978.415,E2 -13978.415} C_VEL
LIN {X 0,Y 500.138,Z 467.365,A -85,B 0,C 180,E1 -13979.062,E2 -13979.062} C_VEL
LIN {X 0,Y 500.808,Z 453.287,A -85,B 0,C 180,E1 -13979.586,E2 -13979.586} C_VEL
LIN {X 0,Y 501.199,Z 438.757,A -85,B 0,C 180,E1 -13979.949,E2 -13979.949} C_VEL
LIN {X 0,Y 502.953,Z 328.212,A -85,B 0,C 180,E1 -13981.568,E2 -13981.568} C_VEL
LIN {X 0,Y 500.642,Z 319.668,A -85,B 0,C 180,E1 -13981.813,E2 -13981.813} C_VEL
LIN {X 0,Y 494.749,Z 304.79,A -85,B 0,C 180,E1 -13982.366,E2 -13982.366} C_VEL
LIN {X 0,Y 492.8,Z 295.657,A -85,B 0,C 180,E1 -13984.474,E2 -13984.474} C_VEL
LIN {X 0,Y 492.775,Z 295.662,A -85,B 0,C 180,E1 -13987.674,E2 -13987.674} C_VEL
LIN {X 0,Y 492.756,Z 295.66,A -85,B 0,C 180,E1 -13990.831,E2 -13990.831} C_VEL
LIN {X 0,Y 492.816,Z 295.658,A -85,B 0,C 180,E1 -13993.542,E2 -13993.542} C_VEL
LIN {X 0,Y 492.816,Z 295.656,A -85,B 0,C 180,E1 -13996.454,E2 -13996.454} C_VEL
LIN {X 0,Y 492.762,Z 295.661,A -85,B 0,C 180,E1 -13999.166,E2 -13999.166} C_VEL
LIN {X 0,Y 492.784,Z 295.655,A -85,B 0,C 180,E1 -14002.323,E2 -14002.323} C_VEL
LIN {X 0,Y 492.818,Z 295.633,A -85,B 0,C 180,E1 -14004.357,E2 -14004.357} C_VEL
LIN {X 0,Y 492.775,Z 295.66,A -85,B 0,C 180,E1 -14007.307,E2 -14007.307} C_VEL
LIN {X 0,Y 492.808,Z 295.656,A -85,B 0,C 180,E1 -14010.167,E2 -14010.167} C_VEL
LIN {X 0,Y 492.818,Z 295.646,A -85,B 0,C 180,E1 -14012.947,E2 -14012.947} C_VEL
LIN {X 0,Y 492.835,Z 295.65,A -85,B 0,C 180,E1 -14015.659,E2 -14015.659} C_VEL
LIN {X 0,Y 492.838,Z 295.65,A -85,B 0,C 180,E1 -14018.314,E2 -14018.314} C_VEL
LIN {X 0,Y 492.831,Z 295.647,A -85,B 0,C 180,E1 -14020.92,E2 -14020.92} C_VEL
LIN {X 0,Y 492.836,Z 295.656,A -85,B 0,C 180,E1 -14023.486,E2 -14023.486} C_VEL
LIN {X 0,Y 492.884,Z 295.637,A -85,B 0,C 180,E1 -14026.02,E2 -14026.02} C_VEL
LIN {X 0,Y 492.948,Z 295.637,A -85,B 0,C 180,E1 -14028.635,E2 -14028.635} C_VEL
LIN {X 0,Y 492.954,Z 295.633,A -85,B 0,C 180,E1 -14031.831,E2 -14031.831} C_VEL
LIN {X 0,Y 493.014,Z 295.627,A -85,B 0,C 180,E1 -14034.292,E2 -14034.292} C_VEL
LIN {X 0,Y 492.976,Z 295.622,A -85,B 0,C 180,E1 -14036.742,E2 -14036.742} C_VEL
LIN {X 0,Y 493.122,Z 295.612,A -85,B 0,C 180,E1 -14040,E2 -14040} C_VEL
LIN {X 0,Y 493.05,Z 295.622,A -85,B 0,C 180,E1 -14044.073,E2 -14044.073} C_VEL
LIN {X 0,Y 493.006,Z 295.627,A -85,B 0,C 180,E1 -14046.526,E2 -14046.526} C_VEL
LIN {X 0,Y 492.939,Z 295.637,A -85,B 0,C 180,E1 -14048.993,E2 -14048.993} C_VEL
LIN {X 0,Y 492.998,Z 295.622,A -85,B 0,C 180,E1 -14051.473,E2 -14051.473} C_VEL
LIN {X 0,Y 492.946,Z 295.639,A -85,B 0,C 180,E1 -14054.942,E2 -14054.942} C_VEL
LIN {X 0,Y 492.873,Z 295.636,A -85,B 0,C 180,E1 -14058.219,E2 -14058.219} C_VEL
LIN {X 0,Y 492.843,Z 295.648,A -85,B 0,C 180,E1 -14060.812,E2 -14060.812} C_VEL
LIN {X 0,Y 492.795,Z 295.653,A -85,B 0,C 180,E1 -14063.452,E2 -14063.452} C_VEL
LIN {X 0,Y 492.823,Z 295.649,A -85,B 0,C 180,E1 -14066.445,E2 -14066.445} C_VEL
LIN {X 0,Y 492.814,Z 295.654,A -85,B 0,C 180,E1 -14068.898,E2 -14068.898} C_VEL
LIN {X 0,Y 492.853,Z 295.647,A -85,B 0,C 180,E1 -14071.725,E2 -14071.725} C_VEL
LIN {X 0,Y 492.819,Z 295.635,A -85,B 0,C 180,E1 -14074.647,E2 -14074.647} C_VEL
LIN {X 0,Y 492.861,Z 295.642,A -85,B 0,C 180,E1 -14077.67,E2 -14077.67} C_VEL
LIN {X 0,Y 492.833,Z 295.653,A -85,B 0,C 180,E1 -14080.827,E2 -14080.827} C_VEL
LIN {X 0,Y 492.823,Z 295.658,A -85,B 0,C 180,E1 -14084.142,E2 -14084.142} C_VEL
LIN {X 0,Y 492.842,Z 295.648,A -85,B 0,C 180,E1 -14086.988,E2 -14086.988} C_VEL
LIN {X 0,Y 492.85,Z 295.655,A -85,B 0,C 180,E1 -14090.245,E2 -14090.245} C_VEL
LIN {X 0,Y 492.853,Z 295.646,A -85,B 0,C 180,E1 -14093.355,E2 -14093.355} C_VEL
LIN {X 0,Y 492.815,Z 295.655,A -85,B 0,C 180,E1 -14096.34,E2 -14096.34} C_VEL
LIN {X 0,Y 492.807,Z 295.663,A -85,B 0,C 180,E1 -14099.227,E2 -14099.227} C_VEL
LIN {X 0,Y 492.834,Z 295.782,A -85,B 0,C 180,E1 -14099.74,E2 -14099.74} C_VEL
LIN {X 0,Y 496.365,Z 310.658,A -85,B 0,C 180,E1 -14102.461,E2 -14102.461} C_VEL
LIN {X 0,Y 498.547,Z 321.865,A -85,B 0,C 180,E1 -14104.406,E2 -14104.406} C_VEL
LIN {X 0,Y 497.09,Z 338.538,A -85,B 0,C 180,E1 -14106.984,E2 -14106.984} C_VEL
LIN {X 0,Y 495.622,Z 356.807,A -85,B 0,C 180,E1 -14109.755,E2 -14109.755} C_VEL
LIN {X 0,Y 500.659,Z 386.457,A -85,B 0,C 180,E1 -14110.456,E2 -14110.456} C_VEL
LIN {X 0,Y 502.016,Z 397.608,A -85,B 0,C 180,E1 -14110.689,E2 -14110.689} C_VEL
LIN {X 0,Y 500.517,Z 495.1,A -85,B 0,C 180,E1 -14112.123,E2 -14112.123} C_VEL
LIN {X 0,Y 499.819,Z 509.389,A -85,B 0,C 180,E1 -14112.485,E2 -14112.485} C_VEL
LIN {X 0,Y 498.975,Z 522.394,A -85,B 0,C 180,E1 -14112.963,E2 -14112.963} C_VEL
LIN {X 0,Y 498.015,Z 534.714,A -85,B 0,C 180,E1 -14113.56,E2 -14113.56} C_VEL
LIN {X 0,Y 496.865,Z 547.628,A -85,B 0,C 180,E1 -14114.361,E2 -14114.361} C_VEL
LIN {X 0,Y 495.717,Z 559.367,A -85,B 0,C 180,E1 -14115.268,E2 -14115.268} C_VEL
LIN {X 0,Y 494.655,Z 570.136,A -85,B 0,C 180,E1 -14116.282,E2 -14116.282} C_VEL
LIN {X 0,Y 493.609,Z 580.822,A -85,B 0,C 180,E1 -14117.504,E2 -14117.504} C_VEL
LIN {X 0,Y 492.901,Z 589.303,A -85,B 0,C 180,E1 -14118.677,E2 -14118.677} C_VEL
LIN {X 0,Y 492.167,Z 597.078,A -85,B 0,C 180,E1 -14119.962,E2 -14119.962} C_VEL
LIN {X 0,Y 491.627,Z 604.186,A -85,B 0,C 180,E1 -14121.399,E2 -14121.399} C_VEL
LIN {X 0,Y 491.292,Z 610.606,A -85,B 0,C 180,E1 -14123.042,E2 -14123.042} C_VEL
LIN {X 0,Y 491.162,Z 616.824,A -85,B 0,C 180,E1 -14124.683,E2 -14124.683} C_VEL
LIN {X 0,Y 491.139,Z 620.466,A -85,B 0,C 180,E1 -14125.913,E2 -14125.913} C_VEL
LIN {X 0,Y 491.114,Z 623.97,A -85,B 0,C 180,E1 -14127.55,E2 -14127.55} C_VEL
LIN {X 0,Y 491.168,Z 625.953,A -85,B 0,C 180,E1 -14129.185,E2 -14129.185} C_VEL
LIN {X 0,Y 491.142,Z 626.454,A -85,B 0,C 180,E1 -14130.819,E2 -14130.819} C_VEL
LIN {X 0,Y 491.099,Z 625.515,A -85,B 0,C 180,E1 -14132.454,E2 -14132.454} C_VEL
LIN {X 0,Y 491.144,Z 623.138,A -85,B 0,C 180,E1 -14134.091,E2 -14134.091} C_VEL
LIN {X 0,Y 491.242,Z 619.269,A -85,B 0,C 180,E1 -14135.73,E2 -14135.73} C_VEL
LIN {X 0,Y 491.483,Z 613.793,A -85,B 0,C 180,E1 -14137.371,E2 -14137.371} C_VEL
LIN {X 0,Y 491.851,Z 607.525,A -85,B 0,C 180,E1 -14138.808,E2 -14138.808} C_VEL
LIN {X 0,Y 492.547,Z 599.68,A -85,B 0,C 180,E1 -14140.241,E2 -14140.241} C_VEL
LIN {X 0,Y 493.229,Z 591.186,A -85,B 0,C 180,E1 -14141.512,E2 -14141.512} C_VEL
LIN {X 0,Y 494.018,Z 581.644,A -85,B 0,C 180,E1 -14142.697,E2 -14142.697} C_VEL
LIN {X 0,Y 494.931,Z 570.758,A -85,B 0,C 180,E1 -14143.819,E2 -14143.819} C_VEL
LIN {X 0,Y 495.956,Z 558.749,A -85,B 0,C 180,E1 -14144.834,E2 -14144.834} C_VEL
LIN {X 0,Y 496.848,Z 547.009,A -85,B 0,C 180,E1 -14145.643,E2 -14145.643} C_VEL
LIN {X 0,Y 497.897,Z 533.227,A -85,B 0,C 180,E1 -14146.396,E2 -14146.396} C_VEL
LIN {X 0,Y 498.742,Z 519.488,A -85,B 0,C 180,E1 -14146.971,E2 -14146.971} C_VEL
LIN {X 0,Y 499.458,Z 504.853,A -85,B 0,C 180,E1 -14147.411,E2 -14147.411} C_VEL
LIN {X 0,Y 502.659,Z 397.784,A -85,B 0,C 180,E1 -14149.445,E2 -14149.445} C_VEL
LIN {X 0,Y 500.727,Z 378.452,A -85,B 0,C 180,E1 -14149.972,E2 -14149.972} C_VEL
LIN {X 0,Y 497.064,Z 354.9,A -85,B 0,C 180,E1 -14150.719,E2 -14150.719} C_VEL
LIN {X 0,Y 495.088,Z 339.105,A -85,B 0,C 180,E1 -14151.584,E2 -14151.584} C_VEL
LIN {X 0,Y 496.52,Z 320.281,A -85,B 0,C 180,E1 -14154.372,E2 -14154.372} C_VEL
LIN {X 0,Y 496.767,Z 315.924,A -85,B 0,C 180,E1 -14155.026,E2 -14155.026} C_VEL
LIN {X 0,Y 493.366,Z 297.977,A -85,B 0,C 180,E1 -14157.939,E2 -14157.939} C_VEL
LIN {X 0,Y 492.869,Z 295.646,A -85,B 0,C 180,E1 -14158.331,E2 -14158.331} C_VEL
LIN {X 0,Y 492.778,Z 295.664,A -85,B 0,C 180,E1 -14161.477,E2 -14161.477} C_VEL
LIN {X 0,Y 492.813,Z 295.656,A -85,B 0,C 180,E1 -14164.649,E2 -14164.649} C_VEL
LIN {X 0,Y 492.756,Z 295.665,A -85,B 0,C 180,E1 -14167.681,E2 -14167.681} C_VEL
LIN {X 0,Y 492.773,Z 295.66,A -85,B 0,C 180,E1 -14170.835,E2 -14170.835} C_VEL
LIN {X 0,Y 492.825,Z 295.653,A -85,B 0,C 180,E1 -14173.543,E2 -14173.543} C_VEL
LIN {X 0,Y 492.83,Z 295.653,A -85,B 0,C 180,E1 -14176.458,E2 -14176.458} C_VEL
LIN {X 0,Y 492.773,Z 295.663,A -85,B 0,C 180,E1 -14179.167,E2 -14179.167} C_VEL
LIN {X 0,Y 492.799,Z 295.658,A -85,B 0,C 180,E1 -14182.325,E2 -14182.325} C_VEL
LIN {X 0,Y 492.827,Z 295.653,A -85,B 0,C 180,E1 -14185.353,E2 -14185.353} C_VEL
LIN {X 0,Y 492.82,Z 295.656,A -85,B 0,C 180,E1 -14188.517,E2 -14188.517} C_VEL
LIN {X 0,Y 492.839,Z 295.652,A -85,B 0,C 180,E1 -14191.104,E2 -14191.104} C_VEL
LIN {X 0,Y 492.832,Z 295.655,A -85,B 0,C 180,E1 -14193.858,E2 -14193.858} C_VEL
LIN {X 0,Y 492.824,Z 295.662,A -85,B 0,C 180,E1 -14196.549,E2 -14196.549} C_VEL
LIN {X 0,Y 492.885,Z 295.658,A -85,B 0,C 180,E1 -14199.711,E2 -14199.711} C_VEL
LIN {X 0,Y 492.877,Z 295.651,A -85,B 0,C 180,E1 -14202.636,E2 -14202.636} C_VEL
LIN {X 0,Y 492.884,Z 295.716,A -85,B 0,C 180,E1 -14203.673,E2 -14203.673} C_VEL
LIN {X 0,Y 496.573,Z 308.526,A -85,B 0,C 180,E1 -14205.917,E2 -14205.917} C_VEL
LIN {X 0,Y 499.148,Z 320.348,A -85,B 0,C 180,E1 -14207.849,E2 -14207.849} C_VEL
LIN {X 0,Y 499.378,Z 324.503,A -85,B 0,C 180,E1 -14208.47,E2 -14208.47} C_VEL
LIN {X 0,Y 498.31,Z 343.028,A -85,B 0,C 180,E1 -14211.105,E2 -14211.105} C_VEL
LIN {X 0,Y 498.208,Z 345.103,A -85,B 0,C 180,E1 -14211.371,E2 -14211.371} C_VEL
LIN {X 0,Y 502.875,Z 366.942,A -85,B 0,C 180,E1 -14212.134,E2 -14212.134} C_VEL
LIN {X 0,Y 503.741,Z 372.442,A -85,B 0,C 180,E1 -14212.303,E2 -14212.303} C_VEL
LIN {X 0,Y 500.315,Z 484.708,A -85,B 0,C 180,E1 -14214.422,E2 -14214.422} C_VEL
LIN {X 0,Y 499.738,Z 498.346,A -85,B 0,C 180,E1 -14214.824,E2 -14214.824} C_VEL
LIN {X 0,Y 498.863,Z 512.79,A -85,B 0,C 180,E1 -14215.419,E2 -14215.419} C_VEL
LIN {X 0,Y 497.895,Z 526.55,A -85,B 0,C 180,E1 -14216.168,E2 -14216.168} C_VEL
LIN {X 0,Y 496.929,Z 538.314,A -85,B 0,C 180,E1 -14216.97,E2 -14216.97} C_VEL
LIN {X 0,Y 495.958,Z 550.358,A -85,B 0,C 180,E1 -14217.977,E2 -14217.977} C_VEL
LIN {X 0,Y 495.116,Z 560.338,A -85,B 0,C 180,E1 -14218.987,E2 -14218.987} C_VEL
LIN {X 0,Y 494.037,Z 570.405,A -85,B 0,C 180,E1 -14220.203,E2 -14220.203} C_VEL
LIN {X 0,Y 493.22,Z 578.725,A -85,B 0,C 180,E1 -14221.424,E2 -14221.424} C_VEL
LIN {X 0,Y 492.439,Z 586.701,A -85,B 0,C 180,E1 -14222.854,E2 -14222.854} C_VEL
LIN {X 0,Y 492.026,Z 592.299,A -85,B 0,C 180,E1 -14224.082,E2 -14224.082} C_VEL
LIN {X 0,Y 491.692,Z 597.461,A -85,B 0,C 180,E1 -14225.507,E2 -14225.507} C_VEL
LIN {X 0,Y 491.462,Z 600.468,A -85,B 0,C 180,E1 -14226.547,E2 -14226.547} C_VEL
LIN {X 0,Y 491.138,Z 603.98,A -85,B 0,C 180,E1 -14228.199,E2 -14228.199} C_VEL
LIN {X 0,Y 491.1,Z 606.008,A -85,B 0,C 180,E1 -14229.855,E2 -14229.855} C_VEL
LIN {X 0,Y 490.94,Z 606.558,A -85,B 0,C 180,E1 -14231.522,E2 -14231.522} C_VEL
LIN {X 0,Y 490.952,Z 605.628,A -85,B 0,C 180,E1 -14233.195,E2 -14233.195} C_VEL
LIN {X 0,Y 491.008,Z 604.58,A -85,B 0,C 180,E1 -14234.054,E2 -14234.054} C_VEL
LIN {X 0,Y 491.035,Z 601.404,A -85,B 0,C 180,E1 -14235.725,E2 -14235.725} C_VEL
LIN {X 0,Y 491.229,Z 597.322,A -85,B 0,C 180,E1 -14237.182,E2 -14237.182} C_VEL
LIN {X 0,Y 491.45,Z 591.651,A -85,B 0,C 180,E1 -14238.704,E2 -14238.704} C_VEL
LIN {X 0,Y 491.784,Z 584.429,A -85,B 0,C 180,E1 -14240.206,E2 -14240.206} C_VEL
LIN {X 0,Y 492.181,Z 576.759,A -85,B 0,C 180,E1 -14241.497,E2 -14241.497} C_VEL
LIN {X 0,Y 492.666,Z 567.401,A -85,B 0,C 180,E1 -14242.794,E2 -14242.794} C_VEL
LIN {X 0,Y 493.253,Z 556.993,A -85,B 0,C 180,E1 -14243.984,E2 -14243.984} C_VEL
LIN {X 0,Y 493.914,Z 545.819,A -85,B 0,C 180,E1 -14245.04,E2 -14245.04} C_VEL
LIN {X 0,Y 494.594,Z 532.785,A -85,B 0,C 180,E1 -14246.041,E2 -14246.041} C_VEL
LIN {X 0,Y 495.268,Z 519.557,A -85,B 0,C 180,E1 -14246.852,E2 -14246.852} C_VEL
LIN {X 0,Y 495.838,Z 506.436,A -85,B 0,C 180,E1 -14247.484,E2 -14247.484} C_VEL
LIN {X 0,Y 496.425,Z 491.861,A -85,B 0,C 180,E1 -14248.008,E2 -14248.008} C_VEL
LIN {X 0,Y 496.747,Z 477.359,A -85,B 0,C 180,E1 -14248.36,E2 -14248.36} C_VEL
LIN {X 0,Y 498.626,Z 369.22,A -85,B 0,C 180,E1 -14250.224,E2 -14250.224} C_VEL
LIN {X 0,Y 495.009,Z 343.297,A -85,B 0,C 180,E1 -14250.816,E2 -14250.816} C_VEL
LIN {X 0,Y 495.858,Z 323.135,A -85,B 0,C 180,E1 -14253.661,E2 -14253.661} C_VEL
LIN {X 0,Y 496.191,Z 312.708,A -85,B 0,C 180,E1 -14255.136,E2 -14255.136} C_VEL
LIN {X 0,Y 492.852,Z 295.652,A -85,B 0,C 180,E1 -14257.735,E2 -14257.735} C_VEL
LIN {X 0,Y 492.796,Z 295.655,A -85,B 0,C 180,E1 -14261.119,E2 -14261.119} C_VEL
LIN {X 0,Y 492.824,Z 295.656,A -85,B 0,C 180,E1 -14264.141,E2 -14264.141} C_VEL
LIN {X 0,Y 492.831,Z 295.651,A -85,B 0,C 180,E1 -14266.982,E2 -14266.982} C_VEL
LIN {X 0,Y 492.799,Z 295.66,A -85,B 0,C 180,E1 -14270.235,E2 -14270.235} C_VEL
LIN {X 0,Y 492.77,Z 295.658,A -85,B 0,C 180,E1 -14273.342,E2 -14273.342} C_VEL
LIN {X 0,Y 492.773,Z 295.663,A -85,B 0,C 180,E1 -14276.332,E2 -14276.332} C_VEL
LIN {X 0,Y 492.799,Z 295.655,A -85,B 0,C 180,E1 -14279.222,E2 -14279.222} C_VEL
LIN {X 0,Y 492.817,Z 295.657,A -85,B 0,C 180,E1 -14282.027,E2 -14282.027} C_VEL
LIN {X 0,Y 492.785,Z 295.657,A -85,B 0,C 180,E1 -14284.758,E2 -14284.758} C_VEL
LIN {X 0,Y 492.865,Z 295.648,A -85,B 0,C 180,E1 -14287.482,E2 -14287.482} C_VEL
LIN {X 0,Y 492.889,Z 295.649,A -85,B 0,C 180,E1 -14290.057,E2 -14290.057} C_VEL
LIN {X 0,Y 492.895,Z 295.643,A -85,B 0,C 180,E1 -14292.635,E2 -14292.635} C_VEL
LIN {X 0,Y 492.939,Z 295.637,A -85,B 0,C 180,E1 -14295.179,E2 -14295.179} C_VEL
LIN {X 0,Y 493.005,Z 295.628,A -85,B 0,C 180,E1 -14298.616,E2 -14298.616} C_VEL
LIN {X 0,Y 493.006,Z 295.724,A -85,B 0,C 180,E1 -14301.522,E2 -14301.522} C_VEL
LIN {X 0,Y 494.536,Z 304.236,A -85,B 0,C 180,E1 -14303.247,E2 -14303.247} C_VEL
LIN {X 0,Y 496.422,Z 311.995,A -85,B 0,C 180,E1 -14303.425,E2 -14303.425} C_VEL
LIN {X 0,Y 499.325,Z 326.424,A -85,B 0,C 180,E1 -14303.732,E2 -14303.732} C_VEL
LIN {X 0,Y 497.98,Z 420.995,A -85,B 0,C 180,E1 -14305.081,E2 -14305.081} C_VEL
LIN {X 0,Y 497.405,Z 426.827,A -85,B 0,C 180,E1 -14305.148,E2 -14305.148} C_VEL
LIN {X 0,Y 492.061,Z 443.808,A -85,B 0,C 180,E1 -14305.299,E2 -14305.299} C_VEL
LIN {X 0,Y 490.819,Z 449.523,A -85,B 0,C 180,E1 -14305.413,E2 -14305.413} C_VEL
LIN {X 0,Y 490.643,Z 451.445,A -85,B 0,C 180,E1 -14305.464,E2 -14305.464} C_VEL
LIN {X 0,Y 490.201,Z 465.127,A -85,B 0,C 180,E1 -14305.952,E2 -14305.952} C_VEL
LIN {X 0,Y 489.61,Z 478.764,A -85,B 0,C 180,E1 -14306.615,E2 -14306.615} C_VEL
LIN {X 0,Y 488.993,Z 491.697,A -85,B 0,C 180,E1 -14307.432,E2 -14307.432} C_VEL
LIN {X 0,Y 488.063,Z 503.505,A -85,B 0,C 180,E1 -14308.353,E2 -14308.353} C_VEL
LIN {X 0,Y 487.432,Z 514.229,A -85,B 0,C 180,E1 -14309.38,E2 -14309.38} C_VEL
LIN {X 0,Y 486.744,Z 523.259,A -85,B 0,C 180,E1 -14310.41,E2 -14310.41} C_VEL
LIN {X 0,Y 486.037,Z 532.327,A -85,B 0,C 180,E1 -14311.65,E2 -14311.65} C_VEL
LIN {X 0,Y 485.553,Z 539.876,A -85,B 0,C 180,E1 -14312.892,E2 -14312.892} C_VEL
LIN {X 0,Y 485.17,Z 546.177,A -85,B 0,C 180,E1 -14314.137,E2 -14314.137} C_VEL
LIN {X 0,Y 484.894,Z 551.354,A -85,B 0,C 180,E1 -14315.386,E2 -14315.386} C_VEL
LIN {X 0,Y 484.531,Z 556.846,A -85,B 0,C 180,E1 -14317.056,E2 -14317.056} C_VEL
LIN {X 0,Y 484.298,Z 559.904,A -85,B 0,C 180,E1 -14318.314,E2 -14318.314} C_VEL
LIN {X 0,Y 484.255,Z 562.756,A -85,B 0,C 180,E1 -14319.993,E2 -14319.993} C_VEL
LIN {X 0,Y 484.173,Z 564.253,A -85,B 0,C 180,E1 -14321.683,E2 -14321.683} C_VEL
LIN {X 0,Y 484.277,Z 564.395,A -85,B 0,C 180,E1 -14323.378,E2 -14323.378} C_VEL
LIN {X 0,Y 484.441,Z 563.171,A -85,B 0,C 180,E1 -14325.083,E2 -14325.083} C_VEL
LIN {X 0,Y 484.701,Z 560.515,A -85,B 0,C 180,E1 -14326.797,E2 -14326.797} C_VEL
LIN {X 0,Y 485.029,Z 557.551,A -85,B 0,C 180,E1 -14328.086,E2 -14328.086} C_VEL
LIN {X 0,Y 485.49,Z 553.655,A -85,B 0,C 180,E1 -14329.378,E2 -14329.378} C_VEL
LIN {X 0,Y 486.038,Z 548.726,A -85,B 0,C 180,E1 -14330.688,E2 -14330.688} C_VEL
LIN {X 0,Y 486.85,Z 541.68,A -85,B 0,C 180,E1 -14332.187,E2 -14332.187} C_VEL
LIN {X 0,Y 487.74,Z 533.896,A -85,B 0,C 180,E1 -14333.527,E2 -14333.527} C_VEL
LIN {X 0,Y 488.706,Z 525.043,A -85,B 0,C 180,E1 -14334.783,E2 -14334.783} C_VEL
LIN {X 0,Y 489.73,Z 515.857,A -85,B 0,C 180,E1 -14335.867,E2 -14335.867} C_VEL
LIN {X 0,Y 490.784,Z 504.904,A -85,B 0,C 180,E1 -14336.942,E2 -14336.942} C_VEL
LIN {X 0,Y 491.851,Z 492.972,A -85,B 0,C 180,E1 -14337.898,E2 -14337.898} C_VEL
LIN {X 0,Y 492.783,Z 480.442,A -85,B 0,C 180,E1 -14338.705,E2 -14338.705} C_VEL
LIN {X 0,Y 493.531,Z 467.245,A -85,B 0,C 180,E1 -14339.373,E2 -14339.373} C_VEL
LIN {X 0,Y 494.207,Z 452.686,A -85,B 0,C 180,E1 -14339.91,E2 -14339.91} C_VEL
LIN {X 0,Y 494.617,Z 438.962,A -85,B 0,C 180,E1 -14340.249,E2 -14340.249} C_VEL
LIN {X 0,Y 496.428,Z 329.537,A -85,B 0,C 180,E1 -14341.872,E2 -14341.872} C_VEL
LIN {X 0,Y 494.476,Z 322.29,A -85,B 0,C 180,E1 -14342.084,E2 -14342.084} C_VEL
LIN {X 0,Y 487.625,Z 305.253,A -85,B 0,C 180,E1 -14342.736,E2 -14342.736} C_VEL
LIN {X 0,Y 485.738,Z 296.536,A -85,B 0,C 180,E1 -14344.792,E2 -14344.792} C_VEL
LIN {X 0,Y 485.753,Z 296.536,A -85,B 0,C 180,E1 -14347.525,E2 -14347.525} C_VEL
LIN {X 0,Y 485.72,Z 296.539,A -85,B 0,C 180,E1 -14350.458,E2 -14350.458} C_VEL
LIN {X 0,Y 485.772,Z 296.535,A -85,B 0,C 180,E1 -14352.661,E2 -14352.661} C_VEL
LIN {X 0,Y 485.759,Z 296.533,A -85,B 0,C 180,E1 -14356.2,E2 -14356.2} C_VEL
LIN {X 0,Y 485.745,Z 296.536,A -85,B 0,C 180,E1 -14358.572,E2 -14358.572} C_VEL
LIN {X 0,Y 485.746,Z 296.539,A -85,B 0,C 180,E1 -14361.68,E2 -14361.68} C_VEL
LIN {X 0,Y 485.751,Z 296.514,A -85,B 0,C 180,E1 -14364.775,E2 -14364.775} C_VEL
LIN {X 0,Y 485.74,Z 296.539,A -85,B 0,C 180,E1 -14367.755,E2 -14367.755} C_VEL
LIN {X 0,Y 485.766,Z 296.531,A -85,B 0,C 180,E1 -14370.642,E2 -14370.642} C_VEL
LIN {X 0,Y 485.785,Z 296.526,A -85,B 0,C 180,E1 -14373.45,E2 -14373.45} C_VEL
LIN {X 0,Y 485.757,Z 296.525,A -85,B 0,C 180,E1 -14376.187,E2 -14376.187} C_VEL
LIN {X 0,Y 485.786,Z 296.529,A -85,B 0,C 180,E1 -14378.871,E2 -14378.871} C_VEL
LIN {X 0,Y 485.816,Z 296.523,A -85,B 0,C 180,E1 -14382.088,E2 -14382.088} C_VEL
LIN {X 0,Y 485.855,Z 296.521,A -85,B 0,C 180,E1 -14384.988,E2 -14384.988} C_VEL
LIN {X 0,Y 485.892,Z 296.515,A -85,B 0,C 180,E1 -14388.357,E2 -14388.357} C_VEL
LIN {X 0,Y 485.914,Z 296.509,A -85,B 0,C 180,E1 -14391.712,E2 -14391.712} C_VEL
LIN {X 0,Y 486.029,Z 296.498,A -85,B 0,C 180,E1 -14395.039,E2 -14395.039} C_VEL
LIN {X 0,Y 485.826,Z 296.523,A -85,B 0,C 180,E1 -14397.521,E2 -14397.521} C_VEL
LIN {X 0,Y 486.077,Z 296.49,A -85,B 0,C 180,E1 -14400,E2 -14400} C_VEL
LIN {X 0,Y 486.014,Z 296.498,A -85,B 0,C 180,E1 -14404.132,E2 -14404.132} C_VEL
LIN {X 0,Y 485.966,Z 296.501,A -85,B 0,C 180,E1 -14406.621,E2 -14406.621} C_VEL
LIN {X 0,Y 485.909,Z 296.515,A -85,B 0,C 180,E1 -14409.124,E2 -14409.124} C_VEL
LIN {X 0,Y 485.94,Z 296.5,A -85,B 0,C 180,E1 -14411.642,E2 -14411.642} C_VEL
LIN {X 0,Y 485.915,Z 296.514,A -85,B 0,C 180,E1 -14415.039,E2 -14415.039} C_VEL
LIN {X 0,Y 485.818,Z 296.517,A -85,B 0,C 180,E1 -14418.493,E2 -14418.493} C_VEL
LIN {X 0,Y 485.786,Z 296.523,A -85,B 0,C 180,E1 -14421.129,E2 -14421.129} C_VEL
LIN {X 0,Y 485.757,Z 296.53,A -85,B 0,C 180,E1 -14423.813,E2 -14423.813} C_VEL
LIN {X 0,Y 485.786,Z 296.525,A -85,B 0,C 180,E1 -14426.631,E2 -14426.631} C_VEL
LIN {X 0,Y 485.779,Z 296.527,A -85,B 0,C 180,E1 -14429.357,E2 -14429.357} C_VEL
LIN {X 0,Y 485.787,Z 296.532,A -85,B 0,C 180,E1 -14432.242,E2 -14432.242} C_VEL
LIN {X 0,Y 485.763,Z 296.508,A -85,B 0,C 180,E1 -14435.224,E2 -14435.224} C_VEL
LIN {X 0,Y 485.816,Z 296.519,A -85,B 0,C 180,E1 -14437.539,E2 -14437.539} C_VEL
LIN {X 0,Y 485.779,Z 296.53,A -85,B 0,C 180,E1 -14440.455,E2 -14440.455} C_VEL
LIN {X 0,Y 485.772,Z 296.532,A -85,B 0,C 180,E1 -14443.87,E2 -14443.87} C_VEL
LIN {X 0,Y 485.802,Z 296.525,A -85,B 0,C 180,E1 -14447.342,E2 -14447.342} C_VEL
LIN {X 0,Y 485.798,Z 296.529,A -85,B 0,C 180,E1 -14450.627,E2 -14450.627} C_VEL
LIN {X 0,Y 485.827,Z 296.521,A -85,B 0,C 180,E1 -14453.841,E2 -14453.841} C_VEL
LIN {X 0,Y 485.782,Z 296.532,A -85,B 0,C 180,E1 -14456.779,E2 -14456.779} C_VEL
LIN {X 0,Y 485.776,Z 296.618,A -85,B 0,C 180,E1 -14459.394,E2 -14459.394} C_VEL
LIN {X 0,Y 489.122,Z 310.556,A -85,B 0,C 180,E1 -14462.002,E2 -14462.002} C_VEL
LIN {X 0,Y 491.718,Z 323.469,A -85,B 0,C 180,E1 -14464.295,E2 -14464.295} C_VEL
LIN {X 0,Y 490.174,Z 339.856,A -85,B 0,C 180,E1 -14466.863,E2 -14466.863} C_VEL
LIN {X 0,Y 488.752,Z 356.189,A -85,B 0,C 180,E1 -14469.392,E2 -14469.392} C_VEL
LIN {X 0,Y 493.331,Z 382.431,A -85,B 0,C 180,E1 -14470.04,E2 -14470.04} C_VEL
LIN {X 0,Y 495.411,Z 397.857,A -85,B 0,C 180,E1 -14470.381,E2 -14470.381} C_VEL
LIN {X 0,Y 493.875,Z 495.147,A -85,B 0,C 180,E1 -14471.837,E2 -14471.837} C_VEL
LIN {X 0,Y 493.144,Z 509.676,A -85,B 0,C 180,E1 -14472.217,E2 -14472.217} C_VEL
LIN {X 0,Y 492.226,Z 522.973,A -85,B 0,C 180,E1 -14472.722,E2 -14472.722} C_VEL
LIN {X 0,Y 491.075,Z 536.831,A -85,B 0,C 180,E1 -14473.427,E2 -14473.427} C_VEL
LIN {X 0,Y 489.901,Z 549.258,A -85,B 0,C 180,E1 -14474.24,E2 -14474.24} C_VEL
LIN {X 0,Y 488.663,Z 561.804,A -85,B 0,C 180,E1 -14475.263,E2 -14475.263} C_VEL
LIN {X 0,Y 487.528,Z 572.096,A -85,B 0,C 180,E1 -14476.289,E2 -14476.289} C_VEL
LIN {X 0,Y 486.526,Z 582.381,A -85,B 0,C 180,E1 -14477.531,E2 -14477.531} C_VEL
LIN {X 0,Y 485.714,Z 591.349,A -85,B 0,C 180,E1 -14478.848,E2 -14478.848} C_VEL
LIN {X 0,Y 484.998,Z 599.107,A -85,B 0,C 180,E1 -14480.232,E2 -14480.232} C_VEL
LIN {X 0,Y 484.419,Z 605.738,A -85,B 0,C 180,E1 -14481.688,E2 -14481.688} C_VEL
LIN {X 0,Y 484.087,Z 616.405,A -85,B 0,C 180,E1 -14484.605,E2 -14484.605} C_VEL
LIN {X 0,Y 484.042,Z 620.114,A -85,B 0,C 180,E1 -14485.853,E2 -14485.853} C_VEL
LIN {X 0,Y 484.026,Z 623.682,A -85,B 0,C 180,E1 -14487.514,E2 -14487.514} C_VEL
LIN {X 0,Y 484.084,Z 625.746,A -85,B 0,C 180,E1 -14489.173,E2 -14489.173} C_VEL
LIN {X 0,Y 484.059,Z 626.316,A -85,B 0,C 180,E1 -14490.831,E2 -14490.831} C_VEL
LIN {X 0,Y 484.012,Z 625.432,A -85,B 0,C 180,E1 -14492.49,E2 -14492.49} C_VEL
LIN {X 0,Y 484.049,Z 623.105,A -85,B 0,C 180,E1 -14494.151,E2 -14494.151} C_VEL
LIN {X 0,Y 484.152,Z 619.297,A -85,B 0,C 180,E1 -14495.814,E2 -14495.814} C_VEL
LIN {X 0,Y 484.442,Z 613.899,A -85,B 0,C 180,E1 -14497.479,E2 -14497.479} C_VEL
LIN {X 0,Y 484.777,Z 608.65,A -85,B 0,C 180,E1 -14498.728,E2 -14498.728} C_VEL
LIN {X 0,Y 485.454,Z 601.156,A -85,B 0,C 180,E1 -14500.182,E2 -14500.182} C_VEL
LIN {X 0,Y 486.229,Z 592.129,A -85,B 0,C 180,E1 -14501.597,E2 -14501.597} C_VEL
LIN {X 0,Y 487.119,Z 582.096,A -85,B 0,C 180,E1 -14502.88,E2 -14502.88} C_VEL
LIN {X 0,Y 488.079,Z 571.319,A -85,B 0,C 180,E1 -14504.017,E2 -14504.017} C_VEL
LIN {X 0,Y 489.15,Z 559.487,A -85,B 0,C 180,E1 -14505.045,E2 -14505.045} C_VEL
LIN {X 0,Y 490.269,Z 546.4,A -85,B 0,C 180,E1 -14505.965,E2 -14505.965} C_VEL
LIN {X 0,Y 491.338,Z 532.495,A -85,B 0,C 180,E1 -14506.727,E2 -14506.727} C_VEL
LIN {X 0,Y 492.182,Z 519.313,A -85,B 0,C 180,E1 -14507.284,E2 -14507.284} C_VEL
LIN {X 0,Y 492.943,Z 504.561,A -85,B 0,C 180,E1 -14507.735,E2 -14507.735} C_VEL
LIN {X 0,Y 496.291,Z 398.432,A -85,B 0,C 180,E1 -14509.801,E2 -14509.801} C_VEL
LIN {X 0,Y 494.486,Z 379.951,A -85,B 0,C 180,E1 -14510.319,E2 -14510.319} C_VEL
LIN {X 0,Y 490.814,Z 356.159,A -85,B 0,C 180,E1 -14511.098,E2 -14511.098} C_VEL
LIN {X 0,Y 488.796,Z 340.76,A -85,B 0,C 180,E1 -14511.932,E2 -14511.932} C_VEL
LIN {X 0,Y 488.345,Z 336.564,A -85,B 0,C 180,E1 -14512.175,E2 -14512.175} C_VEL
LIN {X 0,Y 489.728,Z 318.112,A -85,B 0,C 180,E1 -14514.958,E2 -14514.958} C_VEL
LIN {X 0,Y 489.153,Z 313.507,A -85,B 0,C 180,E1 -14515.693,E2 -14515.693} C_VEL
LIN {X 0,Y 485.806,Z 296.527,A -85,B 0,C 180,E1 -14518.519,E2 -14518.519} C_VEL
LIN {X 0,Y 485.725,Z 296.539,A -85,B 0,C 180,E1 -14521.699,E2 -14521.699} C_VEL
LIN {X 0,Y 485.759,Z 296.535,A -85,B 0,C 180,E1 -14524.723,E2 -14524.723} C_VEL
LIN {X 0,Y 485.723,Z 296.542,A -85,B 0,C 180,E1 -14527.52,E2 -14527.52} C_VEL
LIN {X 0,Y 485.739,Z 296.536,A -85,B 0,C 180,E1 -14530.461,E2 -14530.461} C_VEL
LIN {X 0,Y 485.776,Z 296.53,A -85,B 0,C 180,E1 -14533.8,E2 -14533.8} C_VEL
LIN {X 0,Y 485.777,Z 296.531,A -85,B 0,C 180,E1 -14536.202,E2 -14536.202} C_VEL
LIN {X 0,Y 485.739,Z 296.535,A -85,B 0,C 180,E1 -14539.541,E2 -14539.541} C_VEL
LIN {X 0,Y 485.801,Z 296.531,A -85,B 0,C 180,E1 -14542.73,E2 -14542.73} C_VEL
LIN {X 0,Y 485.767,Z 296.532,A -85,B 0,C 180,E1 -14545.781,E2 -14545.781} C_VEL
LIN {X 0,Y 485.768,Z 296.534,A -85,B 0,C 180,E1 -14548.728,E2 -14548.728} C_VEL
LIN {X 0,Y 485.796,Z 296.528,A -85,B 0,C 180,E1 -14551.588,E2 -14551.588} C_VEL
LIN {X 0,Y 485.766,Z 296.538,A -85,B 0,C 180,E1 -14554.368,E2 -14554.368} C_VEL
LIN {X 0,Y 485.794,Z 296.535,A -85,B 0,C 180,E1 -14557.34,E2 -14557.34} C_VEL
LIN {X 0,Y 485.854,Z 296.534,A -85,B 0,C 180,E1 -14559.757,E2 -14559.757} C_VEL
LIN {X 0,Y 485.825,Z 296.529,A -85,B 0,C 180,E1 -14563.025,E2 -14563.025} C_VEL
LIN {X 0,Y 485.861,Z 296.741,A -85,B 0,C 180,E1 -14563.188,E2 -14563.188} C_VEL
LIN {X 0,Y 489.721,Z 309.621,A -85,B 0,C 180,E1 -14565.505,E2 -14565.505} C_VEL
LIN {X 0,Y 492.547,Z 322.616,A -85,B 0,C 180,E1 -14567.683,E2 -14567.683} C_VEL
LIN {X 0,Y 492.764,Z 326.762,A -85,B 0,C 180,E1 -14568.313,E2 -14568.313} C_VEL
LIN {X 0,Y 491.68,Z 345.188,A -85,B 0,C 180,E1 -14570.946,E2 -14570.946} C_VEL
LIN {X 0,Y 496.483,Z 367.657,A -85,B 0,C 180,E1 -14571.763,E2 -14571.763} C_VEL
LIN {X 0,Y 497.379,Z 373.949,A -85,B 0,C 180,E1 -14571.955,E2 -14571.955} C_VEL
LIN {X 0,Y 493.766,Z 485.931,A -85,B 0,C 180,E1 -14574.122,E2 -14574.122} C_VEL
LIN {X 0,Y 493.084,Z 500.169,A -85,B 0,C 180,E1 -14574.568,E2 -14574.568} C_VEL
LIN {X 0,Y 492.2,Z 513.78,A -85,B 0,C 180,E1 -14575.153,E2 -14575.153} C_VEL
LIN {X 0,Y 491.221,Z 527.33,A -85,B 0,C 180,E1 -14575.912,E2 -14575.912} C_VEL
LIN {X 0,Y 490.09,Z 540.348,A -85,B 0,C 180,E1 -14576.825,E2 -14576.825} C_VEL
LIN {X 0,Y 489.079,Z 552.008,A -85,B 0,C 180,E1 -14577.845,E2 -14577.845} C_VEL
LIN {X 0,Y 488.088,Z 562.617,A -85,B 0,C 180,E1 -14578.972,E2 -14578.972} C_VEL
LIN {X 0,Y 486.978,Z 572.298,A -85,B 0,C 180,E1 -14580.206,E2 -14580.206} C_VEL
LIN {X 0,Y 486.18,Z 580.334,A -85,B 0,C 180,E1 -14581.445,E2 -14581.445} C_VEL
LIN {X 0,Y 485.365,Z 588.052,A -85,B 0,C 180,E1 -14582.895,E2 -14582.895} C_VEL
LIN {X 0,Y 484.979,Z 593.405,A -85,B 0,C 180,E1 -14584.141,E2 -14584.141} C_VEL
LIN {X 0,Y 484.562,Z 599.044,A -85,B 0,C 180,E1 -14585.807,E2 -14585.807} C_VEL
LIN {X 0,Y 484.183,Z 603.103,A -85,B 0,C 180,E1 -14587.481,E2 -14587.481} C_VEL
LIN {X 0,Y 484.001,Z 605.609,A -85,B 0,C 180,E1 -14589.16,E2 -14589.16} C_VEL
LIN {X 0,Y 483.991,Z 606.438,A -85,B 0,C 180,E1 -14590.22,E2 -14590.22} C_VEL
LIN {X 0,Y 483.841,Z 606.654,A -85,B 0,C 180,E1 -14591.693,E2 -14591.693} C_VEL
LIN {X 0,Y 483.862,Z 605.52,A -85,B 0,C 180,E1 -14593.392,E2 -14593.392} C_VEL
LIN {X 0,Y 483.925,Z 604.393,A -85,B 0,C 180,E1 -14594.245,E2 -14594.245} C_VEL
LIN {X 0,Y 483.923,Z 602.876,A -85,B 0,C 180,E1 -14595.102,E2 -14595.102} C_VEL
LIN {X 0,Y 484.042,Z 599.796,A -85,B 0,C 180,E1 -14596.39,E2 -14596.39} C_VEL
LIN {X 0,Y 484.16,Z 595.743,A -85,B 0,C 180,E1 -14597.687,E2 -14597.687} C_VEL
LIN {X 0,Y 484.421,Z 590.626,A -85,B 0,C 180,E1 -14598.986,E2 -14598.986} C_VEL
LIN {X 0,Y 484.748,Z 583.101,A -85,B 0,C 180,E1 -14600.512,E2 -14600.512} C_VEL
LIN {X 0,Y 485.182,Z 575.113,A -85,B 0,C 180,E1 -14601.823,E2 -14601.823} C_VEL
LIN {X 0,Y 485.743,Z 565.399,A -85,B 0,C 180,E1 -14603.138,E2 -14603.138} C_VEL
LIN {X 0,Y 486.358,Z 554.479,A -85,B 0,C 180,E1 -14604.346,E2 -14604.346} C_VEL
LIN {X 0,Y 487.027,Z 543.071,A -85,B 0,C 180,E1 -14605.385,E2 -14605.385} C_VEL
LIN {X 0,Y 487.703,Z 530.494,A -85,B 0,C 180,E1 -14606.323,E2 -14606.323} C_VEL
LIN {X 0,Y 488.377,Z 516.53,A -85,B 0,C 180,E1 -14607.155,E2 -14607.155} C_VEL
LIN {X 0,Y 489.015,Z 502.191,A -85,B 0,C 180,E1 -14607.802,E2 -14607.802} C_VEL
LIN {X 0,Y 489.59,Z 487.217,A -85,B 0,C 180,E1 -14608.288,E2 -14608.288} C_VEL
LIN {X 0,Y 489.925,Z 471.633,A -85,B 0,C 180,E1 -14608.617,E2 -14608.617} C_VEL
LIN {X 0,Y 491.799,Z 370.384,A -85,B 0,C 180,E1 -14610.394,E2 -14610.394} C_VEL
LIN {X 0,Y 488.044,Z 343.357,A -85,B 0,C 180,E1 -14611.026,E2 -14611.026} C_VEL
LIN {X 0,Y 488.917,Z 322.675,A -85,B 0,C 180,E1 -14613.968,E2 -14613.968} C_VEL
LIN {X 0,Y 489.125,Z 313.469,A -85,B 0,C 180,E1 -14615.286,E2 -14615.286} C_VEL
LIN {X 0,Y 485.795,Z 296.532,A -85,B 0,C 180,E1 -14617.878,E2 -14617.878} C_VEL
LIN {X 0,Y 485.743,Z 296.539,A -85,B 0,C 180,E1 -14620.459,E2 -14620.459} C_VEL
LIN {X 0,Y 485.796,Z 296.53,A -85,B 0,C 180,E1 -14622.662,E2 -14622.662} C_VEL
LIN {X 0,Y 485.774,Z 296.535,A -85,B 0,C 180,E1 -14626.134,E2 -14626.134} C_VEL
LIN {X 0,Y 485.759,Z 296.536,A -85,B 0,C 180,E1 -14628.575,E2 -14628.575} C_VEL
LIN {X 0,Y 485.722,Z 296.537,A -85,B 0,C 180,E1 -14631.676,E2 -14631.676} C_VEL
LIN {X 0,Y 485.734,Z 296.536,A -85,B 0,C 180,E1 -14634.772,E2 -14634.772} C_VEL
LIN {X 0,Y 485.729,Z 296.538,A -85,B 0,C 180,E1 -14637.752,E2 -14637.752} C_VEL
LIN {X 0,Y 485.789,Z 296.53,A -85,B 0,C 180,E1 -14640.642,E2 -14640.642} C_VEL
